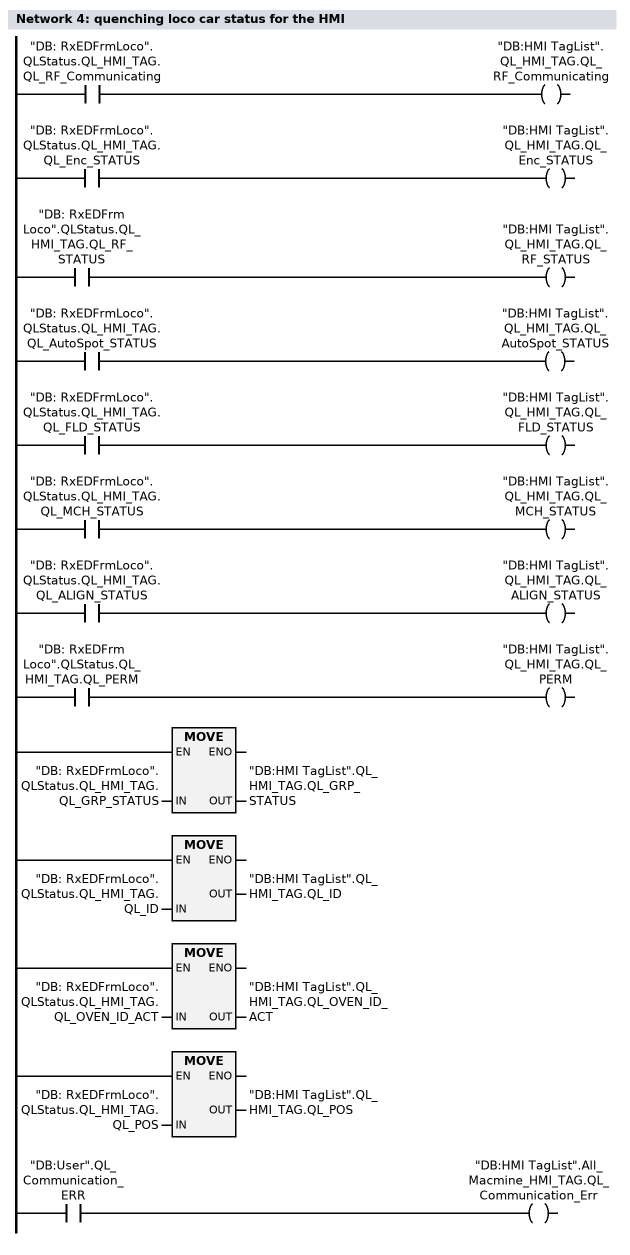
NETWORK
TITLE = quenching loco car status for the HMI
      A     "DB: RxEDFrmLoco".QLStatus.QL_HMI_TAG.QL_RF_Communicating;
      =     "DB:HMI TagList".QL_HMI_TAG.QL_RF_Communicating;
//..
      A     "DB: RxEDFrmLoco".QLStatus.QL_HMI_TAG.QL_Enc_STATUS;
      =     "DB:HMI TagList".QL_HMI_TAG.QL_Enc_STATUS;
//..
      A     "DB: RxEDFrmLoco".QLStatus.QL_HMI_TAG.QL_RF_STATUS;
      =     "DB:HMI TagList".QL_HMI_TAG.QL_RF_STATUS;
//..
      A     "DB: RxEDFrmLoco".QLStatus.QL_HMI_TAG.QL_AutoSpot_STATUS;
      =     "DB:HMI TagList".QL_HMI_TAG.QL_AutoSpot_STATUS;
//..
      A     "DB: RxEDFrmLoco".QLStatus.QL_HMI_TAG.QL_FLD_STATUS;
      =     "DB:HMI TagList".QL_HMI_TAG.QL_FLD_STATUS;
//..
      A     "DB: RxEDFrmLoco".QLStatus.QL_HMI_TAG.QL_MCH_STATUS;
      =     "DB:HMI TagList".QL_HMI_TAG.QL_MCH_STATUS;
//...
      A     "DB: RxEDFrmLoco".QLStatus.QL_HMI_TAG.QL_ALIGN_STATUS;
      =     "DB:HMI TagList".QL_HMI_TAG.QL_ALIGN_STATUS;
//..
      A     "DB: RxEDFrmLoco".QLStatus.QL_HMI_TAG.QL_PERM;
      =     "DB:HMI TagList".QL_HMI_TAG.QL_PERM;
//..
      L     "DB: RxEDFrmLoco".QLStatus.QL_HMI_TAG.QL_GRP_STATUS;
      T     "DB:HMI TagList".QL_HMI_TAG.QL_GRP_STATUS;
//..
      L     "DB: RxEDFrmLoco".QLStatus.QL_HMI_TAG.QL_ID;
      T     "DB:HMI TagList".QL_HMI_TAG.QL_ID;
//...
      L     "DB: RxEDFrmLoco".QLStatus.QL_HMI_TAG.QL_OVEN_ID_ACT;
      T     "DB:HMI TagList".QL_HMI_TAG.QL_OVEN_ID_ACT;
//..
      L     "DB: RxEDFrmLoco".QLStatus.QL_HMI_TAG.QL_POS;
      T     "DB:HMI TagList".QL_HMI_TAG.QL_POS;
//..
      A     "DB:User".QL_Communication_ERR;
      =     "DB:HMI TagList".All_Macmine_HMI_TAG.QL_Communication_Err;
///////////...............
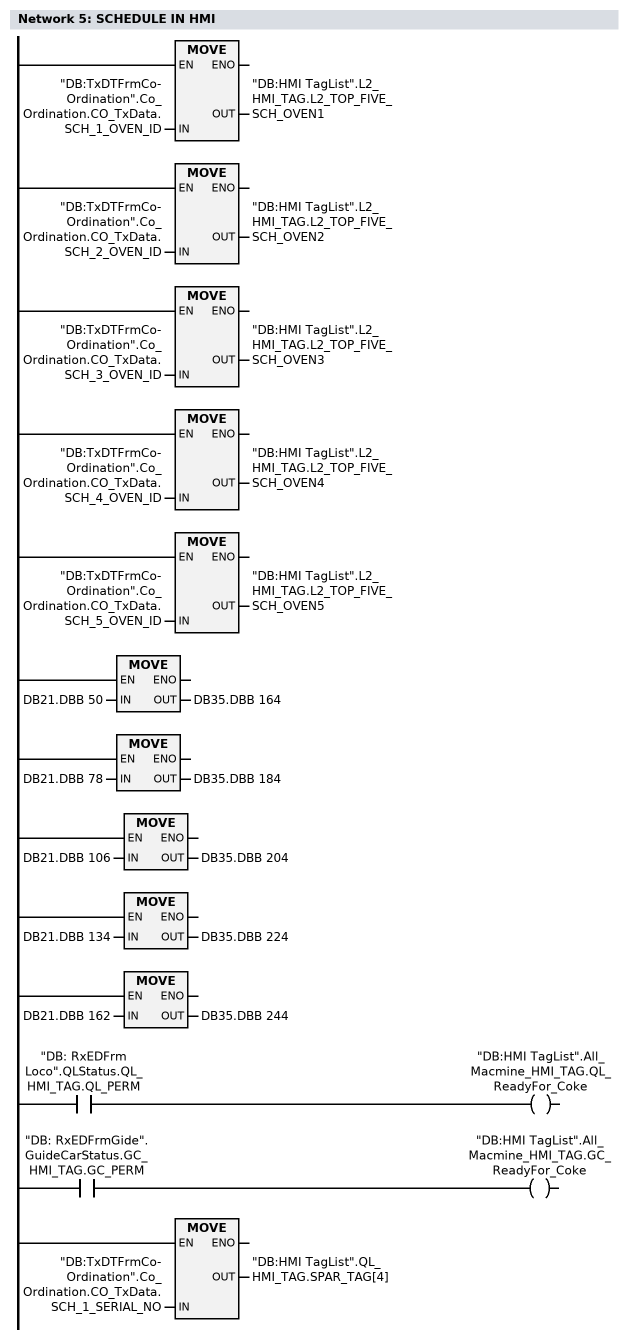
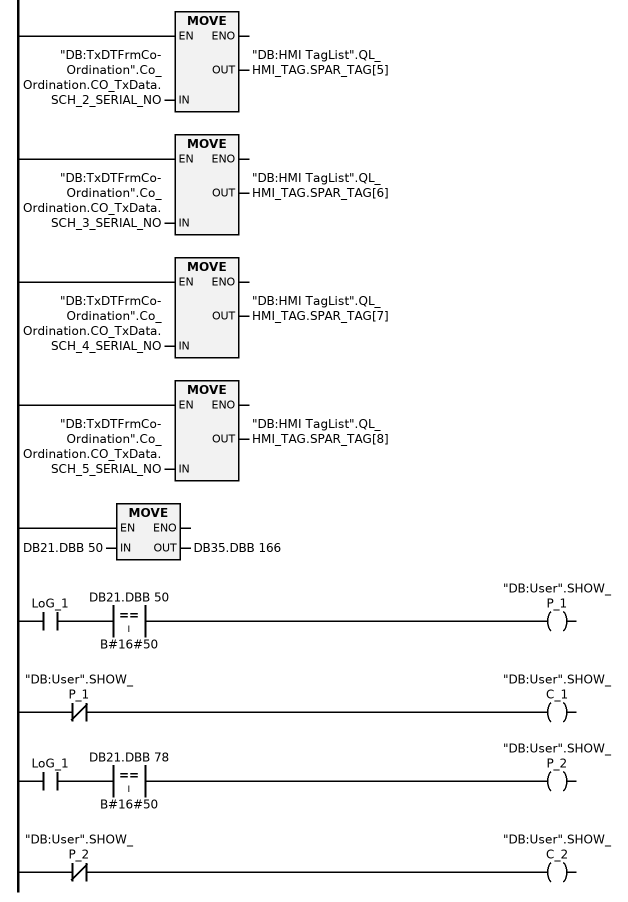
NETWORK
TITLE = SCHEDULE IN HMI
      L     "DB:TxDTFrmCo-Ordination".Co_Ordination.CO_TxData.SCH_1_OVEN_ID;
      T     "DB:HMI TagList".L2_HMI_TAG.L2_TOP_FIVE_SCH_OVEN1;
//..
      L     "DB:TxDTFrmCo-Ordination".Co_Ordination.CO_TxData.SCH_2_OVEN_ID;
      T     "DB:HMI TagList".L2_HMI_TAG.L2_TOP_FIVE_SCH_OVEN2;
//..
      L     "DB:TxDTFrmCo-Ordination".Co_Ordination.CO_TxData.SCH_3_OVEN_ID;
      T     "DB:HMI TagList".L2_HMI_TAG.L2_TOP_FIVE_SCH_OVEN3;
//..
      L     "DB:TxDTFrmCo-Ordination".Co_Ordination.CO_TxData.SCH_4_OVEN_ID;
      T     "DB:HMI TagList".L2_HMI_TAG.L2_TOP_FIVE_SCH_OVEN4;
//..
      L     "DB:TxDTFrmCo-Ordination".Co_Ordination.CO_TxData.SCH_5_OVEN_ID;
      T     "DB:HMI TagList".L2_HMI_TAG.L2_TOP_FIVE_SCH_OVEN5;
//..
      L     DB21.DBB 50;
      T     DB35.DBB 164;
//..
      L     DB21.DBB 78;
      T     DB35.DBB 184;
//..
      L     DB21.DBB 106;
      T     DB35.DBB 204;
//..
      L     DB21.DBB 134;
      T     DB35.DBB 224;
//..
      L     DB21.DBB 162;
      T     DB35.DBB 244;
//...
//...--------QL AND GC PERMISS MOVE TO HMI---------//......
      A     "DB: RxEDFrmLoco".QLStatus.QL_HMI_TAG.QL_PERM;
      =     "DB:HMI TagList".All_Macmine_HMI_TAG.QL_ReadyFor_Coke;
//..
      A     "DB: RxEDFrmGide".GuideCarStatus.GC_HMI_TAG.GC_PERM;
      =     "DB:HMI TagList".All_Macmine_HMI_TAG.GC_ReadyFor_Coke;
//..-------------START OVEEN NO INDICATION TO HMI-----------------------...//
      L     "DB:TxDTFrmCo-Ordination".Co_Ordination.CO_TxData.SCH_1_SERIAL_NO;
      T     "DB:HMI TagList".QL_HMI_TAG.SPAR_TAG[4];
//..
      L     "DB:TxDTFrmCo-Ordination".Co_Ordination.CO_TxData.SCH_2_SERIAL_NO;
      T     "DB:HMI TagList".QL_HMI_TAG.SPAR_TAG[5];
//..
      L     "DB:TxDTFrmCo-Ordination".Co_Ordination.CO_TxData.SCH_3_SERIAL_NO;
      T     "DB:HMI TagList".QL_HMI_TAG.SPAR_TAG[6];
//..
      L     "DB:TxDTFrmCo-Ordination".Co_Ordination.CO_TxData.SCH_4_SERIAL_NO;
      T     "DB:HMI TagList".QL_HMI_TAG.SPAR_TAG[7];
//..
      L     "DB:TxDTFrmCo-Ordination".Co_Ordination.CO_TxData.SCH_5_SERIAL_NO;
      T     "DB:HMI TagList".QL_HMI_TAG.SPAR_TAG[8];
//..
      L     DB21.DBB 50;
      T     DB35.DBB 166;
//..-------------END OVEEN NO INDICATION TO HMI-----------------------...//
//..    show P&C indication for oven no 1&2 in schedule
      A     "LoG_1";
      A(;
      L     DB21.DBB 50;
      L     B#16#50;
      ==I;
      );
      =     "DB:User".SHOW_P_1;
//.. show c indication if not p
      AN    "DB:User".SHOW_P_1;
      =     "DB:User".SHOW_C_1;
//..show P&C indication for oven no 2 in schedule
      A     "LoG_1";
      A(;
      L     DB21.DBB 78;
      L     B#16#50;
      ==I;
      );
      =     "DB:User".SHOW_P_2;
//..
      AN    "DB:User".SHOW_P_2;
      =     "DB:User".SHOW_C_2;
//...========================END===========================================
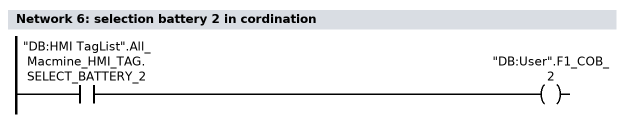
NETWORK
TITLE = selection battery 2 in cordination
      A     "DB:HMI TagList".All_Macmine_HMI_TAG.SELECT_BATTERY_2;
      =     "DB:User".F1_COB_2;
END_FUNCTION

FUNCTION "FC:FreqChanging" : VOID	// FC 28
VERSION : 0.1
VAR_INPUT
  F1_Set : BOOL ;	//Frequency Satting F1 Battery#1
  Offline : BOOL ;	//Machine Offline Mode
END_VAR
VAR_OUTPUT
  ModemFreQ_Set_Don : BOOL ;	//Modem Frequency Set OK
  ModemFreQ_Set_Err : BOOL ;	//Modem Frequency not Set
END_VAR
BEGIN
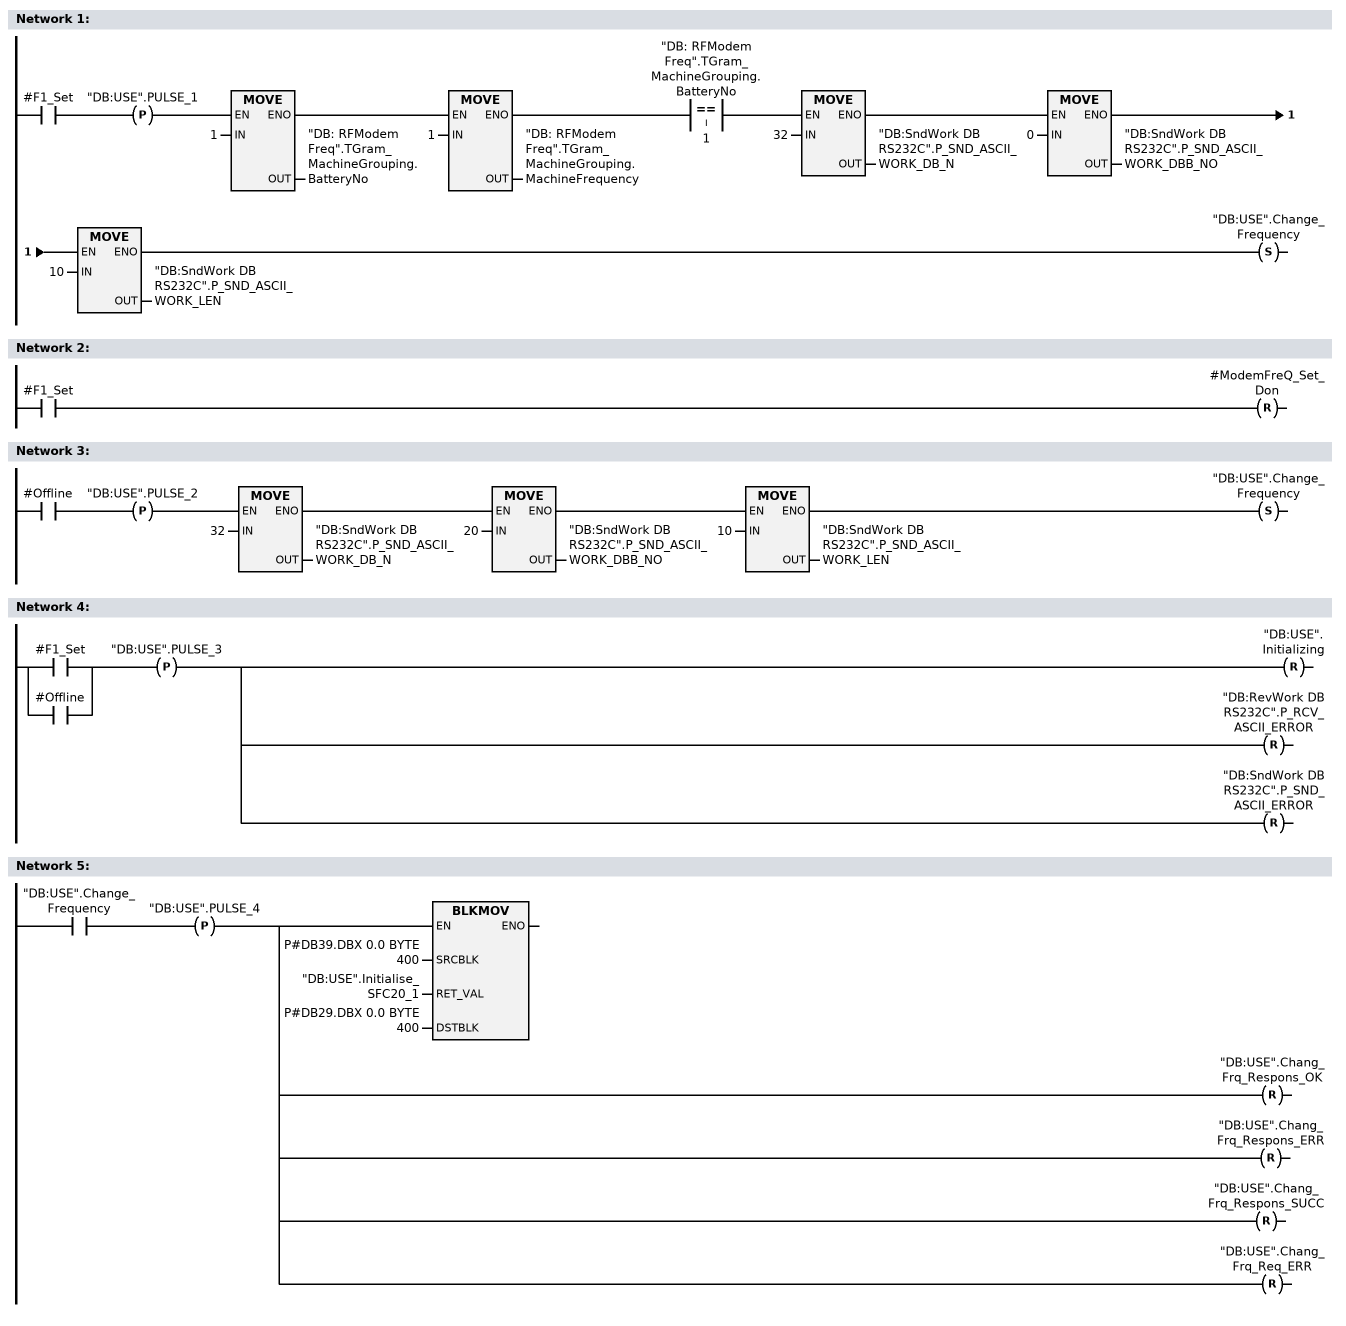
NETWORK
TITLE =
//Change Frequency Request: Initializing        
      A(;
      A(;
      A(;
      A(;
      A     #F1_Set;
      FP    "DB:USE".PULSE_1;
      JNB   _001;
      L     1;
      T     "DB: RFModem Freq".TGram_MachineGrouping.BatteryNo;
      SET;
      SAVE;
      CLR;
_001: A     BR;
      );
      JNB   _002;
      L     1;
      T     "DB: RFModem Freq".TGram_MachineGrouping.MachineFrequency;
      SET;
      SAVE;
      CLR;
_002: A     BR;
      );
      A(;
      L     "DB: RFModem Freq".TGram_MachineGrouping.BatteryNo;
      L     1;
      ==I;
      );
      JNB   _003;
      L     32;
      T     "DB:SndWork DB RS232C".P_SND_ASCII_WORK_DB_N;
      SET;
      SAVE;
      CLR;
_003: A     BR;
      );
      JNB   _004;
      L     0;
      T     "DB:SndWork DB RS232C".P_SND_ASCII_WORK_DBB_NO;
      SET;
      SAVE;
      CLR;
_004: A     BR;
      );
      JNB   _005;
      L     10;
      T     "DB:SndWork DB RS232C".P_SND_ASCII_WORK_LEN;
      SET;
      SAVE;
      CLR;
_005: A     BR;
      S     "DB:USE".Change_Frequency;
NETWORK
TITLE =
      A     #F1_Set;
      R     #ModemFreQ_Set_Don;
NETWORK
TITLE =
//Change Frequency Request: Initializing  
      A(;
      A(;
      A     #Offline;
      FP    "DB:USE".PULSE_2;
      JNB   _006;
      L     32;
      T     "DB:SndWork DB RS232C".P_SND_ASCII_WORK_DB_N;
      SET;
      SAVE;
      CLR;
_006: A     BR;
      );
      JNB   _007;
      L     20;
      T     "DB:SndWork DB RS232C".P_SND_ASCII_WORK_DBB_NO;
      SET;
      SAVE;
      CLR;
_007: A     BR;
      );
      JNB   _008;
      L     10;
      T     "DB:SndWork DB RS232C".P_SND_ASCII_WORK_LEN;
      SET;
      SAVE;
      CLR;
_008: A     BR;
      S     "DB:USE".Change_Frequency;
NETWORK
TITLE =
//Change Frequency Request: Initializing
      A(;
      O     #F1_Set;
      O     #Offline;
      );
      FP    "DB:USE".PULSE_3;
      R     "DB:USE".Initializing;
      R     "DB:RevWork DB RS232C".P_RCV_ASCII_ERROR;
      R     "DB:SndWork DB RS232C".P_SND_ASCII_ERROR;
NETWORK
TITLE =
//Change Frequency Request: Clearing Response Area & ACK/NACK
      A     "DB:USE".Change_Frequency;
      FP    "DB:USE".PULSE_4;
      =     L 0.0;
      A     L 0.0;
      JNB   _009;
      CALL  "BLKMOV" (
           SRCBLK                   := P#DB39.DBX 0.0 BYTE 400,
           RET_VAL                  := "DB:USE".Initialise_SFC20_1,
           DSTBLK                   := P#DB29.DBX 0.0 BYTE 400);
_009: NOP   0;
      A     L 0.0;
      BLD   102;
      R     "DB:USE".Chang_Frq_Respons_OK;
      A     L 0.0;
      BLD   102;
      R     "DB:USE".Chang_Frq_Respons_ERR;
      A     L 0.0;
      BLD   102;
      R     "DB:USE".Chang_Frq_Respons_SUCC;
      A     L 0.0;
      BLD   102;
      R     "DB:USE".Chang_Frq_Req_ERR;
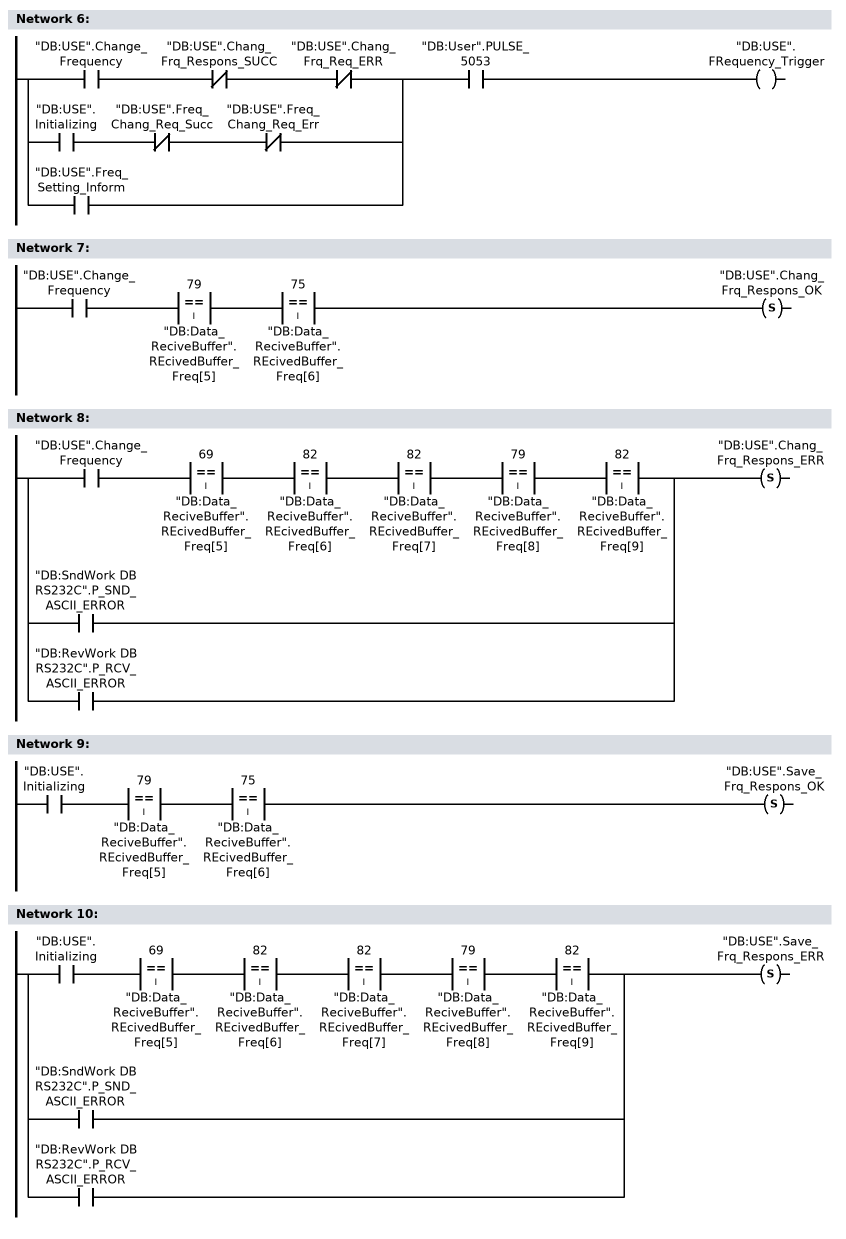
NETWORK
TITLE =
//Change Frequency Request: Try Sending To CP
      A(;
      A     "DB:USE".Change_Frequency;
      AN    "DB:USE".Chang_Frq_Respons_SUCC;
      AN    "DB:USE".Chang_Frq_Req_ERR;
      O;
      A     "DB:USE".Initializing;
      AN    "DB:USE".Freq_Chang_Req_Succ;
      AN    "DB:USE".Freq_Chang_Req_Err;
      O     "DB:USE".Freq_Setting_Inform;
      );
      A     "DB:User".PULSE_5053;
      =     "DB:USE".FRequency_Trigger;
NETWORK
TITLE =
//Change Frequency Request: ACK Response Evaluation (OK Recieved In Empty DB, 
//Succesfull Sent Condition Is Implied Otherwise We Will Not Get Response)
      A     "DB:USE".Change_Frequency;
      A(;
      L     79;	// ASCII 79 = 'O'
      L     "DB:Data_ReciveBuffer".REcivedBuffer_Freq[5];
      ==I;
      );
      A(;
      L     75;	// ASCII 75 = 'K'
      L     "DB:Data_ReciveBuffer".REcivedBuffer_Freq[6];
      ==I;
      );
      S     "DB:USE".Chang_Frq_Respons_OK;
NETWORK
TITLE =
//Change Frequency Request: NACK Response Evaluation (Error Recieved In Empty DB 
//Or Error During Tx Or Rx)
      A     "DB:USE".Change_Frequency;
      A(;
      L     69;	// ASCII 69 = 'E'
      L     "DB:Data_ReciveBuffer".REcivedBuffer_Freq[5];
      ==I;
      );
      A(;
      L     82;	// ASCII 82 = 'R'
      L     "DB:Data_ReciveBuffer".REcivedBuffer_Freq[6];
      ==I;
      );
      A(;
      L     82;	// ASCII 82 = 'R'
      L     "DB:Data_ReciveBuffer".REcivedBuffer_Freq[7];
      ==I;
      );
      A(;
      L     79;	// ASCII 79 = 'O'
      L     "DB:Data_ReciveBuffer".REcivedBuffer_Freq[8];
      ==I;
      );
      A(;
      L     82;	// ASCII 82 = 'R'
      L     "DB:Data_ReciveBuffer".REcivedBuffer_Freq[9];
      ==I;
      );
      O     "DB:SndWork DB RS232C".P_SND_ASCII_ERROR;
      O     "DB:RevWork DB RS232C".P_RCV_ASCII_ERROR;
      S     "DB:USE".Chang_Frq_Respons_ERR;
NETWORK
TITLE =
//Save Frequency Request: ACK Response Evaluation (OK Recieved In Empty DB, 
//Succesfull Sent Condition Is Implied Otherwise We Will Not Get Response)
      A     "DB:USE".Initializing;
      A(;
      L     79;	// ASCII 79 = 'O'
      L     "DB:Data_ReciveBuffer".REcivedBuffer_Freq[5];
      ==I;
      );
      A(;
      L     75;	// ASCII 75 = 'K'
      L     "DB:Data_ReciveBuffer".REcivedBuffer_Freq[6];
      ==I;
      );
      S     "DB:USE".Save_Frq_Respons_OK;
NETWORK
TITLE =
//Save Frequency Request: NACK Response Evaluation (Error Recieved In Empty DB 
//Or Error During Tx Or Rx)
      A     "DB:USE".Initializing;
      A(;
      L     69;	// ASCII 69 = 'E'
      L     "DB:Data_ReciveBuffer".REcivedBuffer_Freq[5];
      ==I;
      );
      A(;
      L     82;	// ASCII 82 = 'R'
      L     "DB:Data_ReciveBuffer".REcivedBuffer_Freq[6];
      ==I;
      );
      A(;
      L     82;	// ASCII 82 = 'R'
      L     "DB:Data_ReciveBuffer".REcivedBuffer_Freq[7];
      ==I;
      );
      A(;
      L     79;	// ASCII 79 = 'O'
      L     "DB:Data_ReciveBuffer".REcivedBuffer_Freq[8];
      ==I;
      );
      A(;
      L     82;	// ASCII 82 = 'R'
      L     "DB:Data_ReciveBuffer".REcivedBuffer_Freq[9];
      ==I;
      );
      O     "DB:SndWork DB RS232C".P_SND_ASCII_ERROR;
      O     "DB:RevWork DB RS232C".P_RCV_ASCII_ERROR;
      S     "DB:USE".Save_Frq_Respons_ERR;
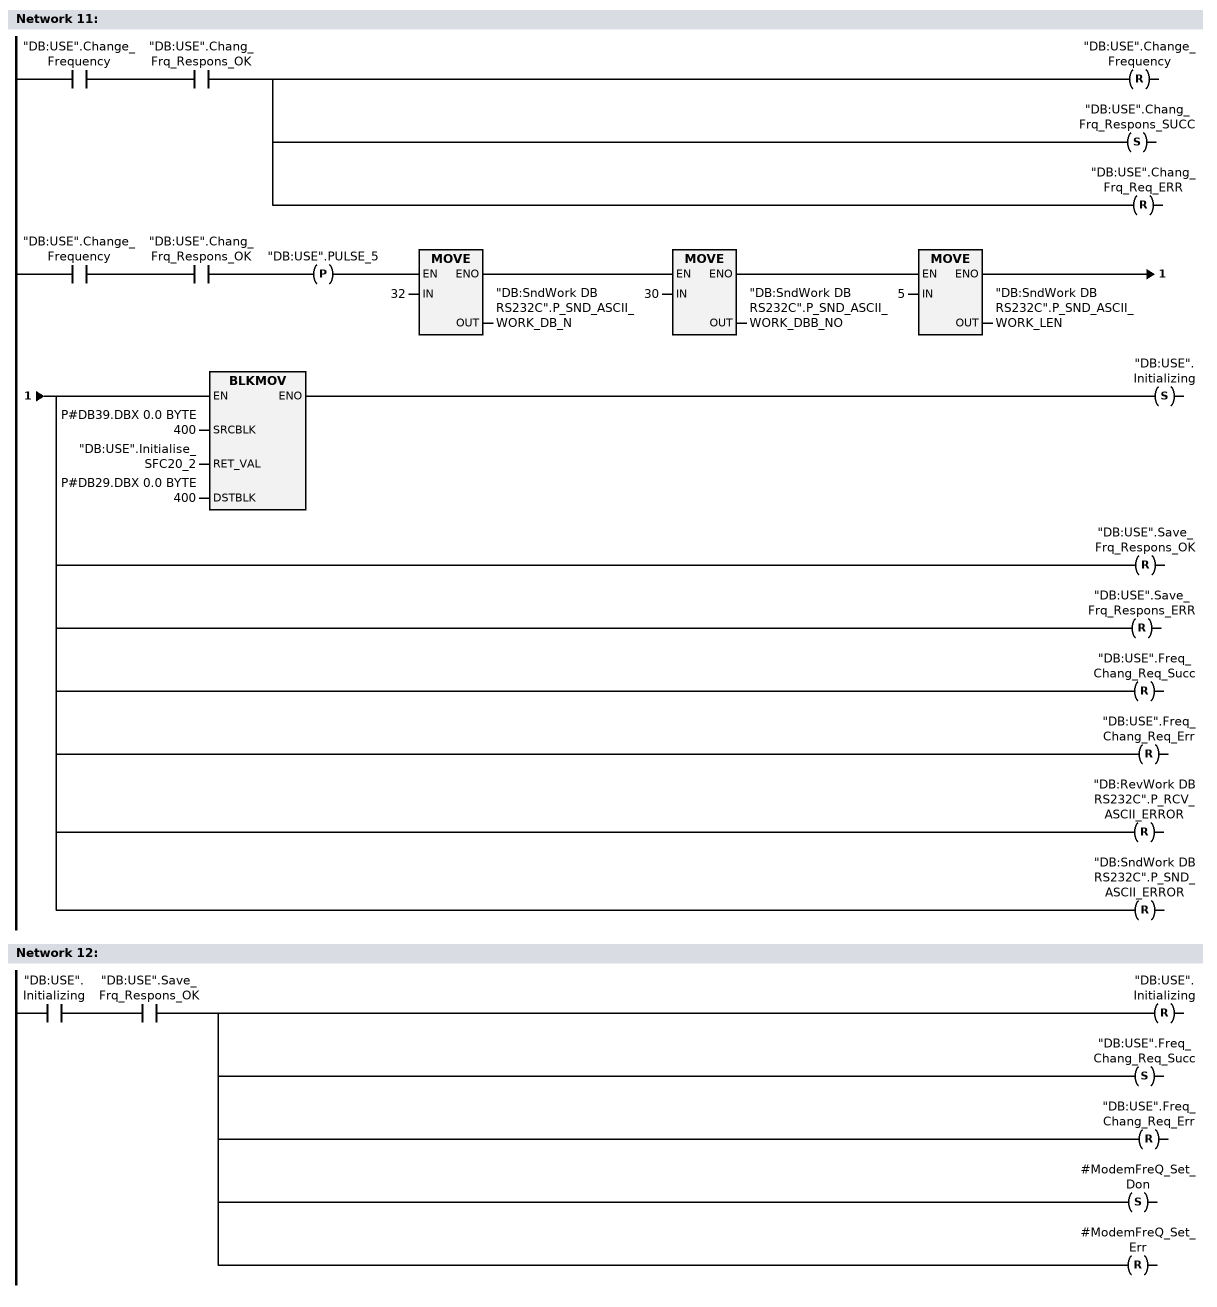
NETWORK
TITLE =
//Change Frequency Request: Success (Sent & ACK Recieved)
      A     "DB:USE".Change_Frequency;
      A     "DB:USE".Chang_Frq_Respons_OK;
      =     L 0.0;
      A     L 0.0;
      BLD   102;
      R     "DB:USE".Change_Frequency;
      A     L 0.0;
      BLD   102;
      S     "DB:USE".Chang_Frq_Respons_SUCC;
      A     L 0.0;
      BLD   102;
      R     "DB:USE".Chang_Frq_Req_ERR;
      A(;
      A(;
      A     L 0.0;
      FP    "DB:USE".PULSE_5;
      JNB   _00a;
      L     32;
      T     "DB:SndWork DB RS232C".P_SND_ASCII_WORK_DB_N;
      SET;
      SAVE;
      CLR;
_00a: A     BR;
      );
      JNB   _00b;
      L     30;
      T     "DB:SndWork DB RS232C".P_SND_ASCII_WORK_DBB_NO;
      SET;
      SAVE;
      CLR;
_00b: A     BR;
      );
      JNB   _00c;
      L     5;
      T     "DB:SndWork DB RS232C".P_SND_ASCII_WORK_LEN;
      SET;
      SAVE;
      CLR;
_00c: A     BR;
      =     L 0.1;
      A     L 0.1;
      JNB   _00d;
      CALL  "BLKMOV" (
           SRCBLK                   := P#DB39.DBX 0.0 BYTE 400,
           RET_VAL                  := "DB:USE".Initialise_SFC20_2,
           DSTBLK                   := P#DB29.DBX 0.0 BYTE 400);
_00d: A     BR;
      S     "DB:USE".Initializing;
      A     L 0.1;
      BLD   102;
      R     "DB:USE".Save_Frq_Respons_OK;
      A     L 0.1;
      BLD   102;
      R     "DB:USE".Save_Frq_Respons_ERR;
      A     L 0.1;
      BLD   102;
      R     "DB:USE".Freq_Chang_Req_Succ;
      A     L 0.1;
      BLD   102;
      R     "DB:USE".Freq_Chang_Req_Err;
      A     L 0.1;
      BLD   102;
      R     "DB:RevWork DB RS232C".P_RCV_ASCII_ERROR;
      A     L 0.1;
      BLD   102;
      R     "DB:SndWork DB RS232C".P_SND_ASCII_ERROR;
NETWORK
TITLE =
//Change Frequency Request: Success (Sent & ACK Recieved)
      A     "DB:USE".Initializing;
      A     "DB:USE".Save_Frq_Respons_OK;
      R     "DB:USE".Initializing;
      S     "DB:USE".Freq_Chang_Req_Succ;
      R     "DB:USE".Freq_Chang_Req_Err;
      S     #ModemFreQ_Set_Don;
      R     #ModemFreQ_Set_Err;
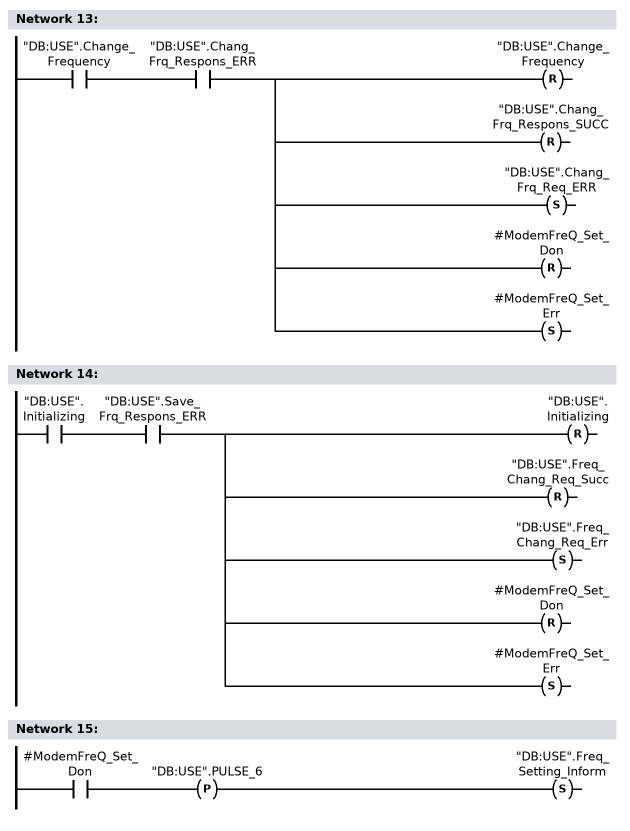
NETWORK
TITLE =
//Change Frequency Request: Error, Or NACK Recieved -> Set Error, Reset Done
      A     "DB:USE".Change_Frequency;
      A     "DB:USE".Chang_Frq_Respons_ERR;
      R     "DB:USE".Change_Frequency;
      R     "DB:USE".Chang_Frq_Respons_SUCC;
      S     "DB:USE".Chang_Frq_Req_ERR;
      R     #ModemFreQ_Set_Don;
      S     #ModemFreQ_Set_Err;
NETWORK
TITLE =
//Save Frequency Request: Error, Or NACK Recieved -> Set Error, Reset Done
      A     "DB:USE".Initializing;
      A     "DB:USE".Save_Frq_Respons_ERR;
      R     "DB:USE".Initializing;
      R     "DB:USE".Freq_Chang_Req_Succ;
      S     "DB:USE".Freq_Chang_Req_Err;
      R     #ModemFreQ_Set_Don;
      S     #ModemFreQ_Set_Err;
NETWORK
TITLE =
//Modem Frequency Set In F1= 436.2 Hz ;
//This Information Sand to Co-Ordination PLC Via RF
      A     #ModemFreQ_Set_Don;
      FP    "DB:USE".PULSE_6;
      S     "DB:USE".Freq_Setting_Inform;
NETWORK
TITLE =
NETWORK
TITLE =
NETWORK
TITLE =
      BE;
END_FUNCTION

FUNCTION "FC:RS232C RCV BLOCK" : VOID	// FC 29
VERSION : 0.1
VAR_INPUT
  CP_BassAdd : INT ;	//LADDR
  DB_No : INT ;	//DB No
  DBB_NO : INT ;	//Data Byte No
END_VAR
BEGIN
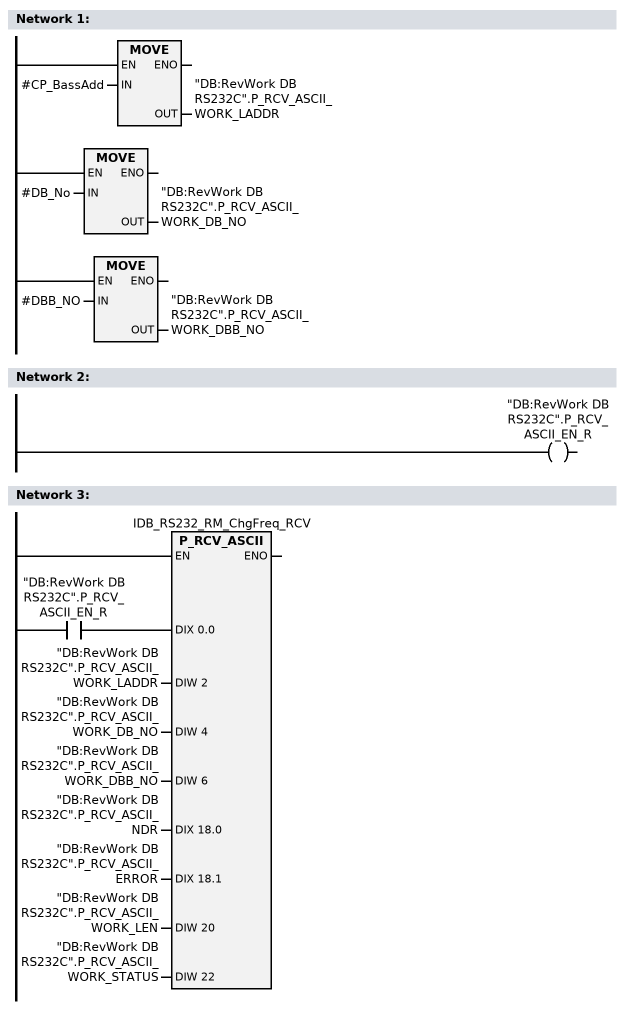
NETWORK
TITLE =
// ----------------------------
// Supply LADDR, DB_NO, DBB_NO
// ----------------------------
      L     #CP_BassAdd;
      T     "DB:RevWork DB RS232C".P_RCV_ASCII_WORK_LADDR;
//..
      L     #DB_No;
      T     "DB:RevWork DB RS232C".P_RCV_ASCII_WORK_DB_NO;
//..
      L     #DBB_NO;
      T     "DB:RevWork DB RS232C".P_RCV_ASCII_WORK_DBB_NO;
NETWORK
TITLE =
//// ------------------------
//// Enable Receive Data
//// ------------------------
//
      SET;
      =     "DB:RevWork DB RS232C".P_RCV_ASCII_EN_R;
NETWORK
TITLE =
//// ------------------------
//// P_RCV_RK with Instance-DB
//// ------------------------
//
      A     "DB:RevWork DB RS232C".P_RCV_ASCII_EN_R;
      =     L 0.0;
      BLD   103;
      CALL  "P_RCV_ASCII" , "IDB_RS232_RM_ChgFreq_RCV" (
           DIX 0.0                  := L 0.0,
           DIW 2                    := "DB:RevWork DB RS232C".P_RCV_ASCII_WORK_LADDR,
           DIW 4                    := "DB:RevWork DB RS232C".P_RCV_ASCII_WORK_DB_NO,
           DIW 6                    := "DB:RevWork DB RS232C".P_RCV_ASCII_WORK_DBB_NO,
           DIX 18.0                 := "DB:RevWork DB RS232C".P_RCV_ASCII_NDR,
           DIX 18.1                 := "DB:RevWork DB RS232C".P_RCV_ASCII_ERROR,
           DIW 20                   := "DB:RevWork DB RS232C".P_RCV_ASCII_WORK_LEN,
           DIW 22                   := "DB:RevWork DB RS232C".P_RCV_ASCII_WORK_STATUS);
      NOP   0;
NETWORK
TITLE =
// -------------------------------
// Check P_RCV_RK_NDR (Receive without error)
// -------------------------------
      AN    "DB:RevWork DB RS232C".P_RCV_ASCII_NDR;	//check P_RCV_RK_NDR
      JC    CHER;	//if P_RCV_RK_NDR equals FALSE, jump to CHER
//and check P_RCV_RK_ERROR
// -------------------------------
//  P_RCV_RK_NDR = 1 (Receive without error)
// -------------------------------
      L     "DB:RevWork DB RS232C".P_RCV_ASCII_WORK_CNT_OK;	//"Receive without error"
      +     1;	//increment counter
      T     "DB:RevWork DB RS232C".P_RCV_ASCII_WORK_CNT_OK;
      L     "DB:RevWork DB RS232C".P_RCV_ASCII_WORK_LEN;	//save RECEIVE-Length
      T     "DB:RevWork DB RS232C".P_RCV_ASCII_WORK_SAVE_LE;
      BE;
// -------------------------------
// Check "Receive with error"
// -------------------------------
CHER: AN    "DB:RevWork DB RS232C".P_RCV_ASCII_ERROR;	//check P_RCV_RK_ERROR
      BEC;	//if no error occured, jump to end
// -------------------------------
// "Receive with error"
// -------------------------------
      L     "DB:RevWork DB RS232C".P_RCV_ASCII_WORK_CNT_ERR;	//Error
      +     1;	//increment counter
      T     "DB:RevWork DB RS232C".P_RCV_ASCII_WORK_CNT_ERR;
// ----------------------------
// Save "P_RCV_RK_STATUS"
// ---------------------------- 
      L     "DB:RevWork DB RS232C".P_RCV_ASCII_WORK_STATUS;
      T     "DB:RevWork DB RS232C".P_RCV_WORK_STATUS_SAV;	//save P_RCV_RK_STATUS
      BE;
END_FUNCTION

FUNCTION "FC:RS232C SND BLOCK" : VOID	// FC 30
TITLE = Execute P_SND_ASCII-Jobs
VERSION : 0.1
VAR_INPUT
  SetFREQ : BOOL ;	//Req
  CP_BassAdd : INT ;	//LADDR
  DB_No : INT ;	//DB No
  DBB_NO : INT ;	//Data Byte No
  LEN : INT ;	//Lenth of Data
END_VAR
BEGIN
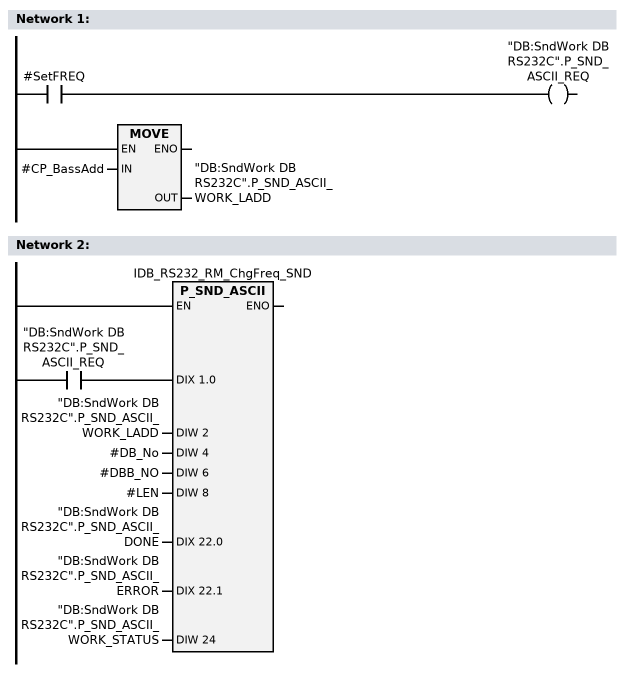
NETWORK
TITLE =
//------------------------
// Supply LADDR, DB_NO, DBB_NO, LEN
// ------------------------
// ------------------------
// Generate edge SEND_REQ
// ------------------------
      A     #SetFREQ;
      =     "DB:SndWork DB RS232C".P_SND_ASCII_REQ;	//Set SEND_REQ
//..
      L     #CP_BassAdd;	//LADDR
      T     "DB:SndWork DB RS232C".P_SND_ASCII_WORK_LADD;
NETWORK
TITLE =
//// ------------------------
//// SEND with Instance-DB
//// ------------------------
//
      A     "DB:SndWork DB RS232C".P_SND_ASCII_REQ;
      =     L 0.0;
      BLD   103;
      CALL  "P_SND_ASCII" , "IDB_RS232_RM_ChgFreq_SND" (
           DIX 1.0                  := L 0.0,
           DIW 2                    := "DB:SndWork DB RS232C".P_SND_ASCII_WORK_LADD,
           DIW 4                    := #DB_No,
           DIW 6                    := #DBB_NO,
           DIW 8                    := #LEN,
           DIX 22.0                 := "DB:SndWork DB RS232C".P_SND_ASCII_DONE,
           DIX 22.1                 := "DB:SndWork DB RS232C".P_SND_ASCII_ERROR,
           DIW 24                   := "DB:SndWork DB RS232C".P_SND_ASCII_WORK_STATUS);
      NOP   0;
NETWORK
TITLE =
// -------------------------------
// Check "Complete without error"
// -------------------------------
      AN    "DB:SndWork DB RS232C".P_SND_ASCII_DONE;	//check P_SND_RK_DONE
      JC    CHER;	//if P_SND_RK_DONE equals 0, jump to CHER
//and check P_SND_RK_ERROR
// -------------------------------
// "Complete without error"
//  P_SND_RK_DONE = 1
// -------------------------------
      L     "DB:SndWork DB RS232C".P_SND_ASCII_COUNTER_OK;	//"Complete without Error"
      +     1;	//increment counter
      T     "DB:SndWork DB RS232C".P_SND_ASCII_COUNTER_OK;
      NOP   0;
      NOP   0;	//further user functions
      NOP   0;
      BE;
// -------------------------------
// Check "Complete with error"
// P_SND_RK_ERROR = 1
// -------------------------------
CHER: AN    "DB:SndWork DB RS232C".P_SND_ASCII_ERROR;	//check P_SND_RK_ERROR
      BEC;	//if no error occured, jump to end
// -------------------------------
// "Complete with error"
// -------------------------------
      L     "DB:SndWork DB RS232C".P_SND_ASCII_COUNTER_ERR;	//"Complete with error"
      +     1;	//increment counter
      T     "DB:SndWork DB RS232C".P_SND_ASCII_COUNTER_ERR;
      L     "DB:SndWork DB RS232C".P_SND_ASCII_WORK_STATUS;
      T     "DB:SndWork DB RS232C".P_SND_WORK_STATUS_SAV;	//save STATUS
      NOP   0;
      NOP   0;	//Error-Handling
      NOP   0;
      BE;
NETWORK
TITLE =
END_FUNCTION

FUNCTION "FC: RdAutoSPOT" : VOID	// FC 31
//This function reads AutoSPOT Telegrams & performs following jobs
//
//1. Detect Packets Recieved, Verify Packets Recieved & Detect No Data 
//(LinkFail). Link fail is a condition when no data or invalid data (except unit 
//id & crc matching) occurs for 8 seconds. Link fail is availaible as function 
//output.
//2. Extract plate address from recieved information packet when aligned and not 
//linkfail and add 100 constant to update oven id output. In case of LinkFail 
//last oven id is retained as output (Note: Same locations like ovens, 
//quenching-towers etc for both batteries shall have different plate number 
//unlike in VSP)
//3. Extract unit id from any packet when not linkfail and update unit id output. 
//In case of LinkFail last unit id is retained as output 
//4. Extract aligned, left aligned and right aligned from any packet recieved and 
//not linkfail
//5. If Detects Machine In Wrong Battery from Currently Selected Battery using 
//Marker Plate Value
//
//Reserved:
//- DB31: AutoSPOT Communication -> Data, Status and Results Are Stored Here
//- DB71: Instance DB for AutoSPOT Communication
//- C127: Timeout Detection Counter
AUTHOR : SKD
NAME : CDSPL
VERSION : 0.1
VAR_INPUT
  Enable : BOOL ;	//Enable AutoSPOT Reading
  CPAddr : INT ;	//Base Address of RS485 Card (CP341)
  SelBatt : INT ;	//Currently Selected Battery {0 - Offline, 1-Battery #1, 2-Battery #2}
END_VAR
VAR_OUTPUT
  OvenID : INT ;	//Oven Number Machine Is Aligned At.
  UnitID : INT ;	//UnitID Of Connected AutoSPOT H/w
  Aligned : BOOL ;	//True = If Both S9/Left & S10/Right Markers Are Blocked
  S9Aligned : BOOL ;	//True = If S9/Left Marker Is Blocked
  S10Aligned : BOOL ;	//True = If S10/Right Marker Is Blocked
  LinkFail : BOOL ;	//True = If Communication Error, Bad Data Etc.
  McInWrongBatt : BOOL ;	//True If Machine Movement In Wrong Battery
END_VAR
VAR_TEMP
  tCtrCV : WORD ;
  tOvenID : INT ;
END_VAR
BEGIN
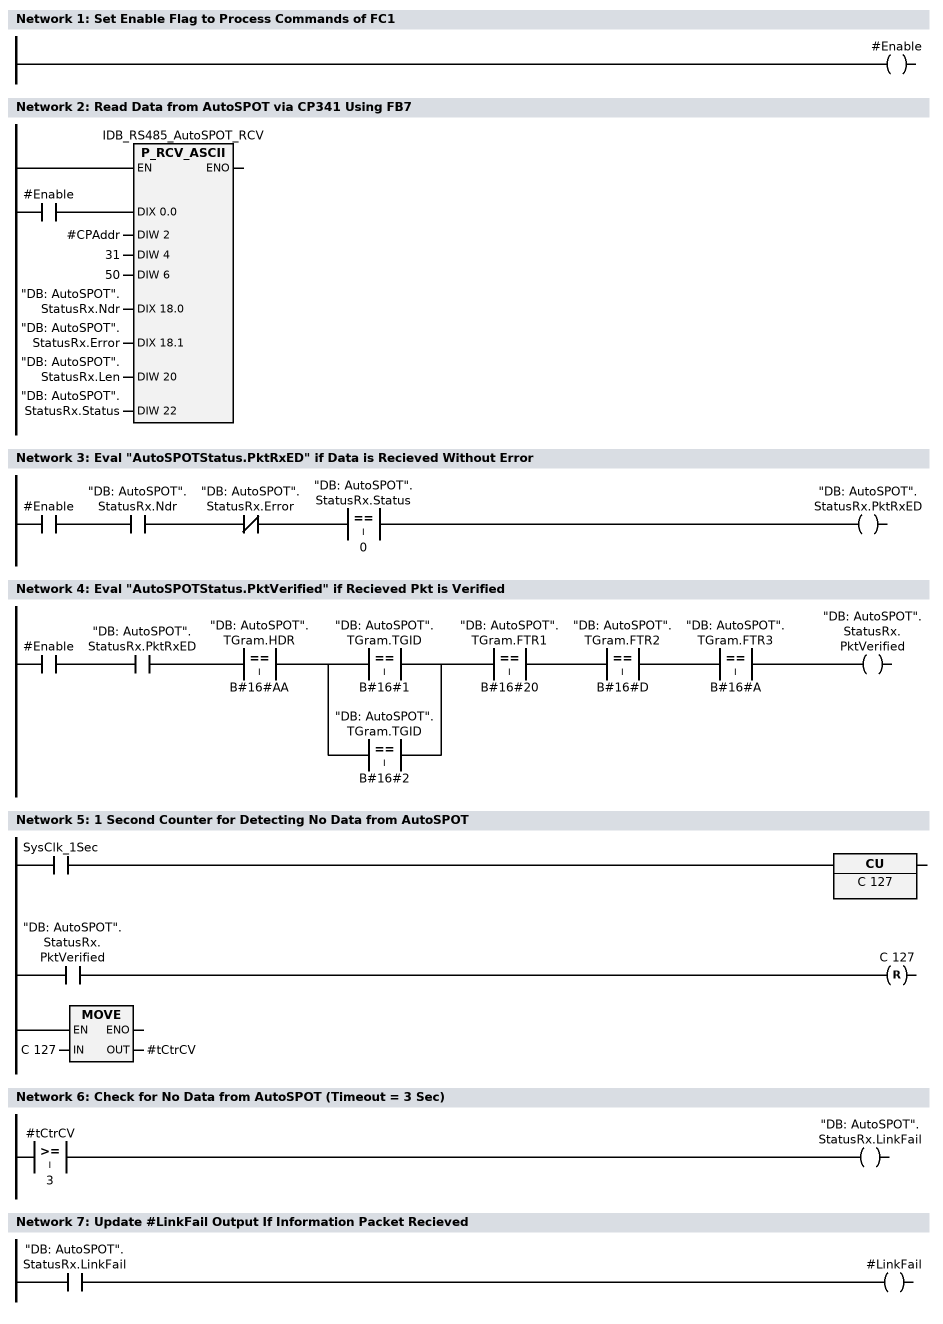
NETWORK
TITLE = Set Enable Flag to Process Commands of FC1
//Set Enable Flag to Process Commands of FC1
      SET;
      =     #Enable;
NETWORK
TITLE = Read Data from AutoSPOT via CP341 Using FB7
//Read Data from AutoSPOT via CP341 Using FB7
      A     #Enable;
      =     L 4.0;
      BLD   103;
      CALL  "P_RCV_ASCII" , "IDB_RS485_AutoSPOT_RCV" (
           DIX 0.0                  := L 4.0,
           DIW 2                    := #CPAddr,
           DIW 4                    := 31,
           DIW 6                    := 50,
           DIX 18.0                 := "DB: AutoSPOT".StatusRx.Ndr,
           DIX 18.1                 := "DB: AutoSPOT".StatusRx.Error,
           DIW 20                   := "DB: AutoSPOT".StatusRx.Len,
           DIW 22                   := "DB: AutoSPOT".StatusRx.Status);
      NOP   0;
NETWORK
TITLE = Eval "AutoSPOTStatus.PktRxED" if Data is Recieved Without Error
//Eval "AutoSPOTStatus.PktRxED" if Data is Recieved Without Error
//(Condition: Ndr And !Error AND Status=0) 
      A     #Enable;
      A     "DB: AutoSPOT".StatusRx.Ndr;
      AN    "DB: AutoSPOT".StatusRx.Error;
      A(;
      L     "DB: AutoSPOT".StatusRx.Status;
      L     0;
      ==I;
      );
      =     "DB: AutoSPOT".StatusRx.PktRxED;
NETWORK
TITLE = Eval "AutoSPOTStatus.PktVerified" if Recieved Pkt is Verified
//Eval "AutoSPOTStatus.PktVerified" if Recieved Pkt is Verified
//(Condition: Match HDR, TGID, & FTR1 to FTR3; Ignore CRC)
      A     #Enable;
      A     "DB: AutoSPOT".StatusRx.PktRxED;
//Match HDR
      A(;
      L     "DB: AutoSPOT".TGram.HDR;
      L     B#16#AA;
      ==I;
      );
//Match TGID
      A(;
      O(;
      L     "DB: AutoSPOT".TGram.TGID;
      L     B#16#1;
      ==I;
      );
      O(;
      L     "DB: AutoSPOT".TGram.TGID;
      L     B#16#2;
      ==I;
      );
      );
//Match FTR1
      A(;
      L     "DB: AutoSPOT".TGram.FTR1;
      L     B#16#20;
      ==I;
      );
//Match FTR2
      A(;
      L     "DB: AutoSPOT".TGram.FTR2;
      L     B#16#D;
      ==I;
      );
//Match FTR3
      A(;
      L     "DB: AutoSPOT".TGram.FTR3;
      L     B#16#A;
      ==I;
      );
      =     "DB: AutoSPOT".StatusRx.PktVerified;
NETWORK
TITLE = 1 Second Counter for Detecting No Data from AutoSPOT
//1 Second Counter for Detecting No Data from AutoSPOT
      A     "SysClk_1Sec";
      CU    C 127;
      BLD   101;
      NOP   0;
      NOP   0;
      A     "DB: AutoSPOT".StatusRx.PktVerified;
      R     C 127;
      L     C 127;
      T     #tCtrCV;
      NOP   0;
      NOP   0;
NETWORK
TITLE = Check for No Data from AutoSPOT (Timeout = 3 Sec)
//Check for No Data from AutoSPOT (Timeout = 3 Sec)
//Match Counter > 3 Seconds
      L     #tCtrCV;
      L     3;
      >=I;
      =     "DB: AutoSPOT".StatusRx.LinkFail;
NETWORK
TITLE = Update #LinkFail Output If Information Packet Recieved
//Update #LinkFail Output If Information Packet Recieved
      A     "DB: AutoSPOT".StatusRx.LinkFail;
      =     #LinkFail;
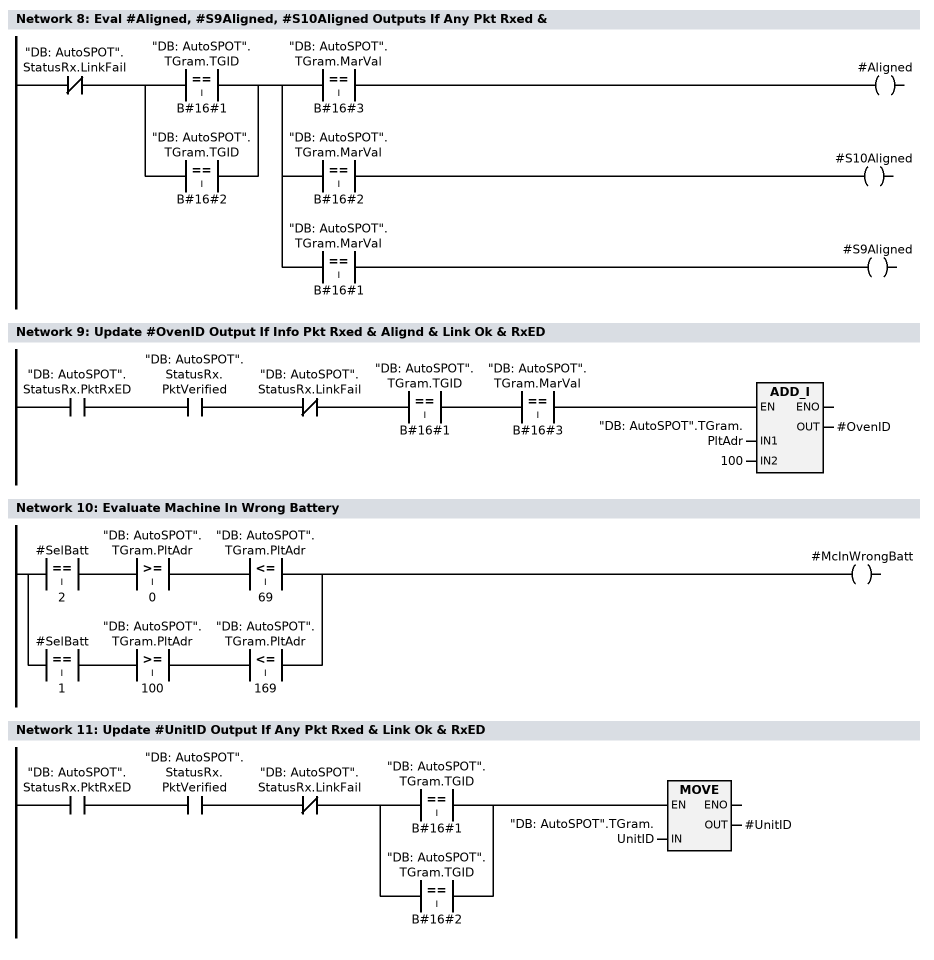
NETWORK
TITLE = Eval #Aligned, #S9Aligned, #S10Aligned Outputs If Any Pkt Rxed &
//Eval #Aligned, #S9Aligned, #S10Aligned Outputs If Any Pkt Rxed & Link Is Ok
      AN    "DB: AutoSPOT".StatusRx.LinkFail;
      A(;
      O(;
      L     "DB: AutoSPOT".TGram.TGID;
      L     B#16#1;
      ==I;
      );
      O(;
      L     "DB: AutoSPOT".TGram.TGID;
      L     B#16#2;
      ==I;
      );
      );
      =     L 2.0;
      A     L 2.0;
      A(;
      L     "DB: AutoSPOT".TGram.MarVal;
      L     B#16#3;
      ==I;
      );
      =     #Aligned;
      A     L 2.0;
      A(;
      L     "DB: AutoSPOT".TGram.MarVal;
      L     B#16#2;
      ==I;
      );
      =     #S10Aligned;
      A     L 2.0;
      A(;
      L     "DB: AutoSPOT".TGram.MarVal;
      L     B#16#1;
      ==I;
      );
      =     #S9Aligned;
NETWORK
TITLE = Update #OvenID Output If Info Pkt Rxed & Alignd & Link Ok & RxED
//Update #OvenID Output If Info Pkt Rxed & Alignd & Link Ok & RxED
      A     "DB: AutoSPOT".StatusRx.PktRxED;
      A     "DB: AutoSPOT".StatusRx.PktVerified;
      AN    "DB: AutoSPOT".StatusRx.LinkFail;
      A(;
      L     "DB: AutoSPOT".TGram.TGID;
      L     B#16#1;
      ==I;
      );
      A(;
      L     "DB: AutoSPOT".TGram.MarVal;
      L     B#16#3;
      ==I;
      );
      JNB   _002;
      L     "DB: AutoSPOT".TGram.PltAdr;
      L     100;
      +I;
      T     #OvenID;
_002: NOP   0;
NETWORK
TITLE = Evaluate Machine In Wrong Battery
//If Selection = Battery #2/1 && PlateValue from #0/100-69/169 => Machine Is 
//Moved In Wrong Battery
      A(;
      L     #SelBatt;
      L     2;
      ==I;
      );
      A(;
      L     "DB: AutoSPOT".TGram.PltAdr;
      L     0;
      >=I;
      );
      A(;
      L     "DB: AutoSPOT".TGram.PltAdr;
      L     69;
      <=I;
      );
      O;
      A(;
      L     #SelBatt;
      L     1;
      ==I;
      );
      A(;
      L     "DB: AutoSPOT".TGram.PltAdr;
      L     100;
      >=I;
      );
      A(;
      L     "DB: AutoSPOT".TGram.PltAdr;
      L     169;
      <=I;
      );
      =     #McInWrongBatt;
NETWORK
TITLE = Update #UnitID Output If Any Pkt Rxed & Link Ok & RxED
//Update #UnitID Output If Any Pkt Rxed & Link Ok & RxED
      A     "DB: AutoSPOT".StatusRx.PktRxED;
      A     "DB: AutoSPOT".StatusRx.PktVerified;
      AN    "DB: AutoSPOT".StatusRx.LinkFail;
      A(;
      O(;
      L     "DB: AutoSPOT".TGram.TGID;
      L     B#16#1;
      ==I;
      );
      O(;
      L     "DB: AutoSPOT".TGram.TGID;
      L     B#16#2;
      ==I;
      );
      );
      JNB   _001;
      L     "DB: AutoSPOT".TGram.UnitID;
      T     #UnitID;
_001: NOP   0;
NETWORK
TITLE = Error Status Handling
//Error Status Handling
// -------------------------------
// Check "Receive without error"
// -------------------------------
      A     "DB: AutoSPOT".StatusRx.Ndr;	//NDR ?
      JCN   CON1;	//if NO
      L     DB31.DBW 18;	//"Receive without error"
      +     1;	//increment counter
      T     DB31.DBW 18;
      L     "DB: AutoSPOT".StatusRx.Len;	//save RECEIVE-Length
      T     DB31.DBW 16;
      JU    LEAV;
// -------------------------------
// Check "Receive with error"
// -------------------------------
CON1: A     "DB: AutoSPOT".StatusRx.Error;	//ERROR ?
      JCN   CON2;	//if NO
      L     DB31.DBW 20;	//"Receive with error"
      +     1;	//increment counter
      T     DB31.DBW 20;
      L     0;
      L     "DB: AutoSPOT".StatusRx.Status;	//if STATUS <> 0
      ==I;
      JC    LEAV;
      T     DB31.DBW 22;	//save STATUS
      JU    LEAV;
// ----------------------------
// Check "Error in STATUS"
// ----------------------------
CON2: L     0;
      L     "DB: AutoSPOT".StatusRx.Status;	//if STATUS <> 0
      ==I;
      JC    LEAV;
      T     DB31.DBW 22;	//save STATUS
LEAV: CLR;
END_FUNCTION

FUNCTION "FC:Group_Change_Info" : VOID	// FC 40
VERSION : 0.1
BEGIN
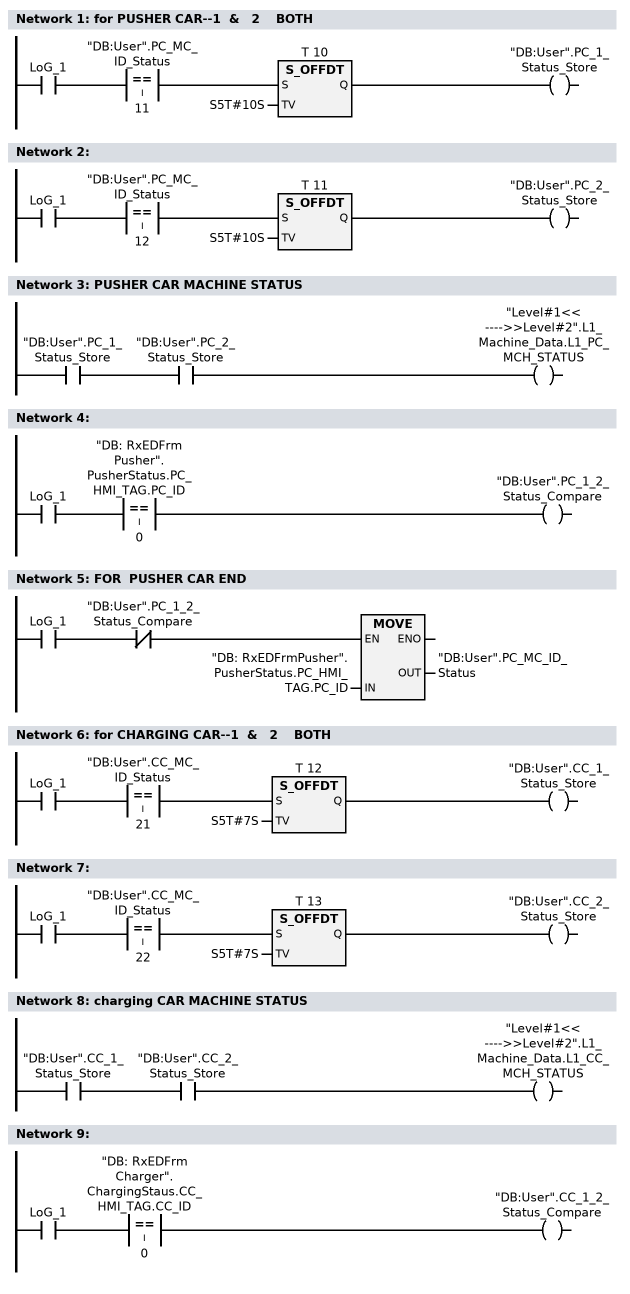
NETWORK
TITLE = for PUSHER CAR--1  &   2    BOTH
//Pusher Car Machine --1 ID Change Over Timer
      A     "LoG_1";
      A(;
      L     "DB:User".PC_MC_ID_Status;
      L     11;
      ==I;
      );
      L     S5T#10S;
      SF    T 10;
      NOP   0;
      NOP   0;
      NOP   0;
      A     T 10;
      =     "DB:User".PC_1_Status_Store;
NETWORK
TITLE =
//Pusher Car Machine --2 ID Change Over Timer
      A     "LoG_1";
      A(;
      L     "DB:User".PC_MC_ID_Status;
      L     12;
      ==I;
      );
      L     S5T#10S;
      SF    T 11;
      NOP   0;
      NOP   0;
      NOP   0;
      A     T 11;
      =     "DB:User".PC_2_Status_Store;
NETWORK
TITLE = PUSHER CAR MACHINE STATUS
//Puser Car Machine Change Over Information Go to L#2
      A     "DB:User".PC_1_Status_Store;
      A     "DB:User".PC_2_Status_Store;
      =     "Level#1<< ---->>Level#2".L1_Machine_Data.L1_PC_MCH_STATUS;
NETWORK
TITLE =
//Pusher Car 1 & 2 Bothe Nachine Compare to Zero Status
      A     "LoG_1";
      A(;
      L     "DB: RxEDFrmPusher".PusherStatus.PC_HMI_TAG.PC_ID;
      L     0;
      ==I;
      );
      =     "DB:User".PC_1_2_Status_Compare;
NETWORK
TITLE = FOR  PUSHER CAR END
//Pusher Car Macine ID Change Information
      A     "LoG_1";
      AN    "DB:User".PC_1_2_Status_Compare;
      JNB   _001;
      L     "DB: RxEDFrmPusher".PusherStatus.PC_HMI_TAG.PC_ID;
      T     "DB:User".PC_MC_ID_Status;
_001: NOP   0;
NETWORK
TITLE = for CHARGING CAR--1  &   2    BOTH
//charging Car Machine --1 ID Change Over Timer
      A     "LoG_1";
      A(;
      L     "DB:User".CC_MC_ID_Status;
      L     21;
      ==I;
      );
      L     S5T#7S;
      SF    T 12;
      NOP   0;
      NOP   0;
      NOP   0;
      A     T 12;
      =     "DB:User".CC_1_Status_Store;
NETWORK
TITLE =
//charging Car Machine --2 ID Change Over Timer
      A     "LoG_1";
      A(;
      L     "DB:User".CC_MC_ID_Status;
      L     22;
      ==I;
      );
      L     S5T#7S;
      SF    T 13;
      NOP   0;
      NOP   0;
      NOP   0;
      A     T 13;
      =     "DB:User".CC_2_Status_Store;
NETWORK
TITLE = charging CAR MACHINE STATUS
//charging Car Machine Change Over Information Go to L#2
      A     "DB:User".CC_1_Status_Store;
      A     "DB:User".CC_2_Status_Store;
      =     "Level#1<< ---->>Level#2".L1_Machine_Data.L1_CC_MCH_STATUS;
NETWORK
TITLE =
//charging Car 1 & 2 Bothe Nachine Compare to Zero Status
      A     "LoG_1";
      A(;
      L     "DB: RxEDFrmCharger".ChargingStaus.CC_HMI_TAG.CC_ID;
      L     0;
      ==I;
      );
      =     "DB:User".CC_1_2_Status_Compare;
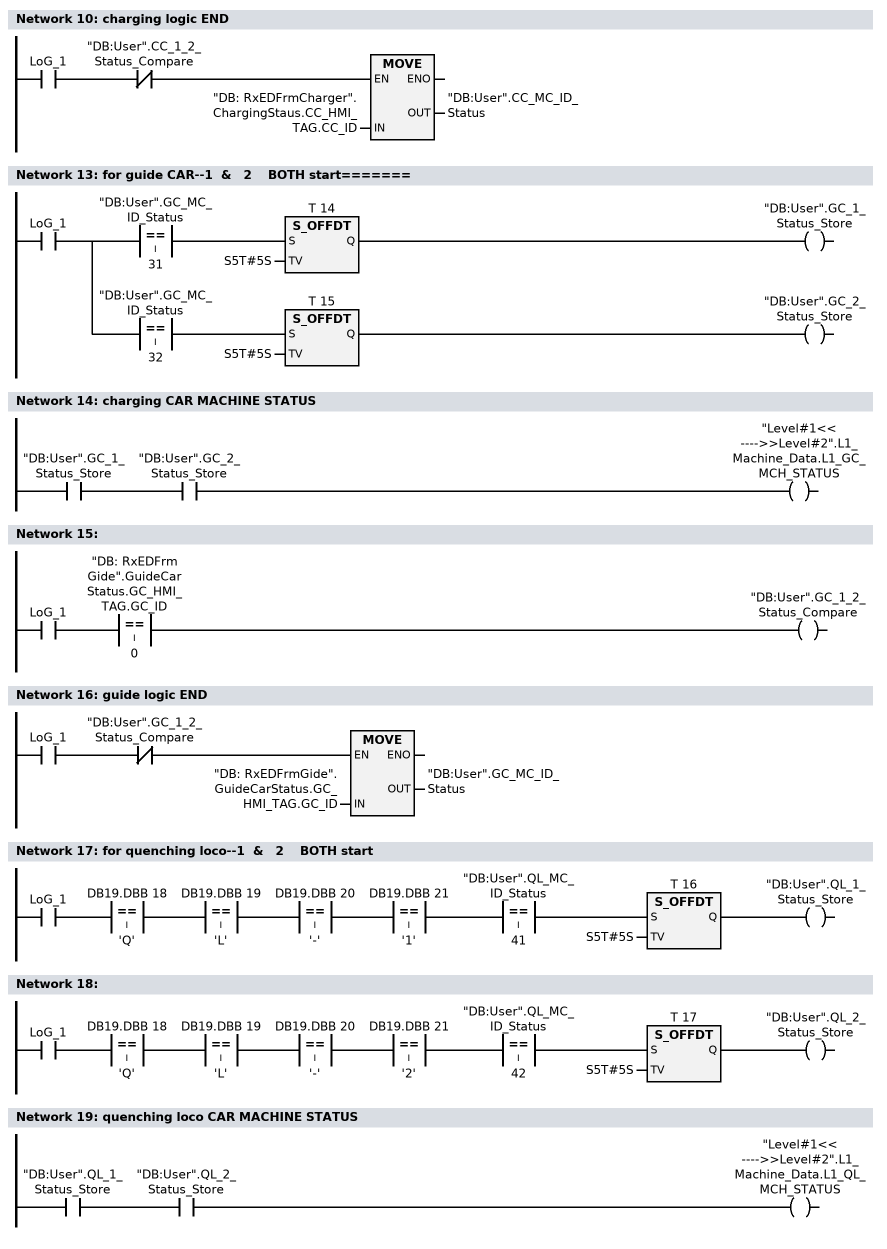
NETWORK
TITLE = charging logic END
//charging Car Macine ID Change Information
      A     "LoG_1";
      AN    "DB:User".CC_1_2_Status_Compare;
      JNB   _002;
      L     "DB: RxEDFrmCharger".ChargingStaus.CC_HMI_TAG.CC_ID;
      T     "DB:User".CC_MC_ID_Status;
_002: NOP   0;
NETWORK
TITLE = for guide CAR--1  &   2    BOTH start
//guide Car Machine --1 ID Change Over Timer
//++++++++++++++++++++++++++++++++++++++++++++++++++++++++++++++++++++++
//
//      A     "LoG_1"
//      A(    
//      L     "DB: RxEDFrmGide".GuideCarStatus.TGInfo.Description[1]
//      L     'G'
//      ==I   
//      )     
//      A(    
//      L     "DB: RxEDFrmGide".GuideCarStatus.TGInfo.Description[2]
//      L     'C'
//      ==I   
//      )     
//      A(    
//      L     "DB: RxEDFrmGide".GuideCarStatus.TGInfo.Description[3]
//      L     '-'
//      ==I   
//      )     
//      A(    
//      L     "DB: RxEDFrmGide".GuideCarStatus.TGInfo.Description[4]
//      L     '1'
//      ==I   
//      )     
//
//      A(    
//      L     "DB:User".GC_MC_ID_Status
//      L     31
//      ==I   
//      )     
//      L     S5T#5S
//      SF    T     14
//      NOP   0
//      NOP   0
//      NOP   0
//      A     T     14
//      =     "DB:User".GC_1_Status_Store
//
NETWORK
TITLE =
//guide Car Machine --2 ID Change Over Timer
//
//++++++++++++++++++++++++++++++++++++++++++++++++++++++
//      A     "LoG_1"
//      A(    
//      L     "DB: RxEDFrmGide".GuideCarStatus.TGInfo.Description[1]
//      L     'G'
//      ==I   
//      )     
//      A(    
//      L     "DB: RxEDFrmGide".GuideCarStatus.TGInfo.Description[2]
//      L     'C'
//      ==I   
//      )     
//      A(    
//      L     "DB: RxEDFrmGide".GuideCarStatus.TGInfo.Description[3]
//      L     '-'
//      ==I   
//      )     
//      A(    
//      L     "DB: RxEDFrmGide".GuideCarStatus.TGInfo.Description[4]
//      L     '2'
//      ==I   
//      )     
//      A(    
//      L     "DB:User".GC_MC_ID_Status
//      L     32
//      ==I   
//      )     
//      L     S5T#5S
//      SF    T     15
//      NOP   0
//      NOP   0
//      NOP   0
//      A     T     15
//      =     "DB:User".GC_2_Status_Store
//
NETWORK
TITLE = for guide CAR--1  &   2    BOTH start=======
      A     "LoG_1";
      =     L 0.0;
      A     L 0.0;
      A(;
      L     "DB:User".GC_MC_ID_Status;
      L     31;
      ==I;
      );
      L     S5T#5S;
      SF    T 14;
      NOP   0;
      NOP   0;
      NOP   0;
      A     T 14;
      =     "DB:User".GC_1_Status_Store;
      A     L 0.0;
      A(;
      L     "DB:User".GC_MC_ID_Status;
      L     32;
      ==I;
      );
      L     S5T#5S;
      SF    T 15;
      NOP   0;
      NOP   0;
      NOP   0;
      A     T 15;
      =     "DB:User".GC_2_Status_Store;
NETWORK
TITLE = charging CAR MACHINE STATUS
//guide Car Machine Change Over Information Go to L#2
      A     "DB:User".GC_1_Status_Store;
      A     "DB:User".GC_2_Status_Store;
      =     "Level#1<< ---->>Level#2".L1_Machine_Data.L1_GC_MCH_STATUS;
NETWORK
TITLE =
//guide Car 1 & 2 Bothe Nachine Compare to Zero Status
      A     "LoG_1";
      A(;
      L     "DB: RxEDFrmGide".GuideCarStatus.GC_HMI_TAG.GC_ID;
      L     0;
      ==I;
      );
      =     "DB:User".GC_1_2_Status_Compare;
NETWORK
TITLE = guide logic END
//guide Car Macine ID Change Information
      A     "LoG_1";
      AN    "DB:User".GC_1_2_Status_Compare;
      JNB   _003;
      L     "DB: RxEDFrmGide".GuideCarStatus.GC_HMI_TAG.GC_ID;
      T     "DB:User".GC_MC_ID_Status;
_003: NOP   0;
NETWORK
TITLE = for quenching loco--1  &   2    BOTH start
//quenching loco Machine --1 ID Change Over Timer
      A     "LoG_1";
      A(;
      L     DB19.DBB 18;
      L     'Q';
      ==I;
      );
      A(;
      L     DB19.DBB 19;
      L     'L';
      ==I;
      );
      A(;
      L     DB19.DBB 20;
      L     '-';
      ==I;
      );
      A(;
      L     DB19.DBB 21;
      L     '1';
      ==I;
      );
      A(;
      L     "DB:User".QL_MC_ID_Status;
      L     41;
      ==I;
      );
      L     S5T#5S;
      SF    T 16;
      NOP   0;
      NOP   0;
      NOP   0;
      A     T 16;
      =     "DB:User".QL_1_Status_Store;
NETWORK
TITLE =
//quenching loco Car Machine --2 ID Change Over Timer
      A     "LoG_1";
      A(;
      L     DB19.DBB 18;
      L     'Q';
      ==I;
      );
      A(;
      L     DB19.DBB 19;
      L     'L';
      ==I;
      );
      A(;
      L     DB19.DBB 20;
      L     '-';
      ==I;
      );
      A(;
      L     DB19.DBB 21;
      L     '2';
      ==I;
      );
      A(;
      L     "DB:User".QL_MC_ID_Status;
      L     42;
      ==I;
      );
      L     S5T#5S;
      SF    T 17;
      NOP   0;
      NOP   0;
      NOP   0;
      A     T 17;
      =     "DB:User".QL_2_Status_Store;
NETWORK
TITLE = quenching loco CAR MACHINE STATUS
//quenching loco Machine Change Over Information Go to L#2
      A     "DB:User".QL_1_Status_Store;
      A     "DB:User".QL_2_Status_Store;
      =     "Level#1<< ---->>Level#2".L1_Machine_Data.L1_QL_MCH_STATUS;
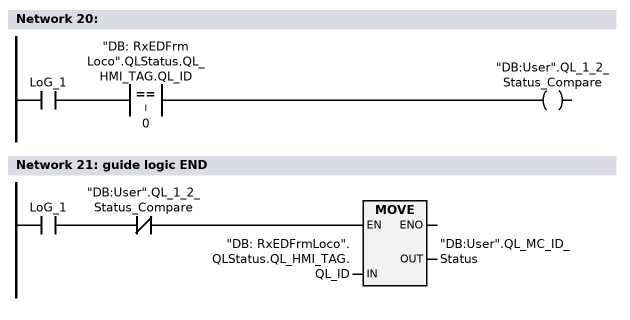
NETWORK
TITLE =
//quenching loco 1 & 2 Bothe Nachine Compare to Zero Status
      A     "LoG_1";
      A(;
      L     "DB: RxEDFrmLoco".QLStatus.QL_HMI_TAG.QL_ID;
      L     0;
      ==I;
      );
      =     "DB:User".QL_1_2_Status_Compare;
NETWORK
TITLE = guide logic END
//guide Car Macine ID Change Information
      A     "LoG_1";
      AN    "DB:User".QL_1_2_Status_Compare;
      JNB   _004;
      L     "DB: RxEDFrmLoco".QLStatus.QL_HMI_TAG.QL_ID;
      T     "DB:User".QL_MC_ID_Status;
_004: NOP   0;
END_FUNCTION

FUNCTION "FC_45_OFFLINE" : VOID	// FC 45
TITLE = moving the data to co-ordination hmi
VERSION : 0.1
VAR_TEMP
  MOV_1 : BOOL ;
  MOV_2 : BOOL ;
  MOV_3 : BOOL ;
  MOV_4 : BOOL ;
  MOV_5 : BOOL ;
  MOV_6 : BOOL ;
  MOV_7 : BOOL ;
  MOV_8 : BOOL ;
  MOV_9 : BOOL ;
  MOV_10 : BOOL ;
  MOV_11 : BOOL ;
  MOV_12 : BOOL ;
  MOV_13 : BOOL ;
  MOV_14 : BOOL ;
  MOV_15 : BOOL ;
  MOV_16 : BOOL ;
  MOV_17 : BOOL ;
  MOV_18 : BOOL ;
  MOV_19 : BOOL ;
  MOV_20 : BOOL ;
  MOV_21 : BOOL ;
  MOV_22 : BOOL ;
  MOV_23 : BOOL ;
  MOV_24 : BOOL ;
  MOV_25 : BOOL ;
  MOV_26 : BOOL ;
  MOV_27 : BOOL ;
  MOV_28 : BOOL ;
  MOV_29 : BOOL ;
  MOV_30 : BOOL ;
  MOV_31 : BOOL ;
  MOV_32 : BOOL ;
  MOV_33 : BOOL ;
  MOV_34 : BOOL ;
  MOV_35 : BOOL ;
  MOV_36 : BOOL ;
  MOV_37 : BOOL ;
  MOV_38 : BOOL ;
  MOV_39 : BOOL ;
  MOV_40 : BOOL ;
  MOV_41 : BOOL ;
  MOV_42 : BOOL ;
  MOV_43 : BOOL ;
  MOV_44 : BOOL ;
  MOV_45 : BOOL ;
  MOV_46 : BOOL ;
  MOV_47 : BOOL ;
  MOV_48 : BOOL ;
  MOV_49 : BOOL ;
  MOV_50 : BOOL ;
  MOV_51 : BOOL ;
  MOV_52 : BOOL ;
  MOV_53 : BOOL ;
  MOV_54 : BOOL ;
  MOV_55 : BOOL ;
  MOV_56 : BOOL ;
  MOV_57 : BOOL ;
  MOV_58 : BOOL ;
  MOV_59 : BOOL ;
  MOV_60 : BOOL ;
  MOV_61 : BOOL ;
  MOV_62 : BOOL ;
  MOV_63 : BOOL ;
  MOV_64 : BOOL ;
  MOV_65 : BOOL ;
  MOV_66 : BOOL ;
  MOV_67 : BOOL ;
  MOV_68 : BOOL ;
  MOV_69 : BOOL ;
  MOV_70 : BOOL ;
  MOV_71 : BOOL ;
  MOV_72 : BOOL ;
  MOV_73 : BOOL ;
  MOV_74 : BOOL ;
  MOV_75 : BOOL ;
  MOV_76 : BOOL ;
  MOV_77 : BOOL ;
  MOV_78 : BOOL ;
  MOV_79 : BOOL ;
  MOV_80 : BOOL ;
  MOV_81 : BOOL ;
  MOV_82 : BOOL ;
  MOV_83 : BOOL ;
  MOV_84 : BOOL ;
  MOV_85 : BOOL ;
  MOV_86 : BOOL ;
  MOV_87 : BOOL ;
  MOV_88 : BOOL ;
  MOV_89 : BOOL ;
  MOV_90 : BOOL ;
END_VAR
BEGIN
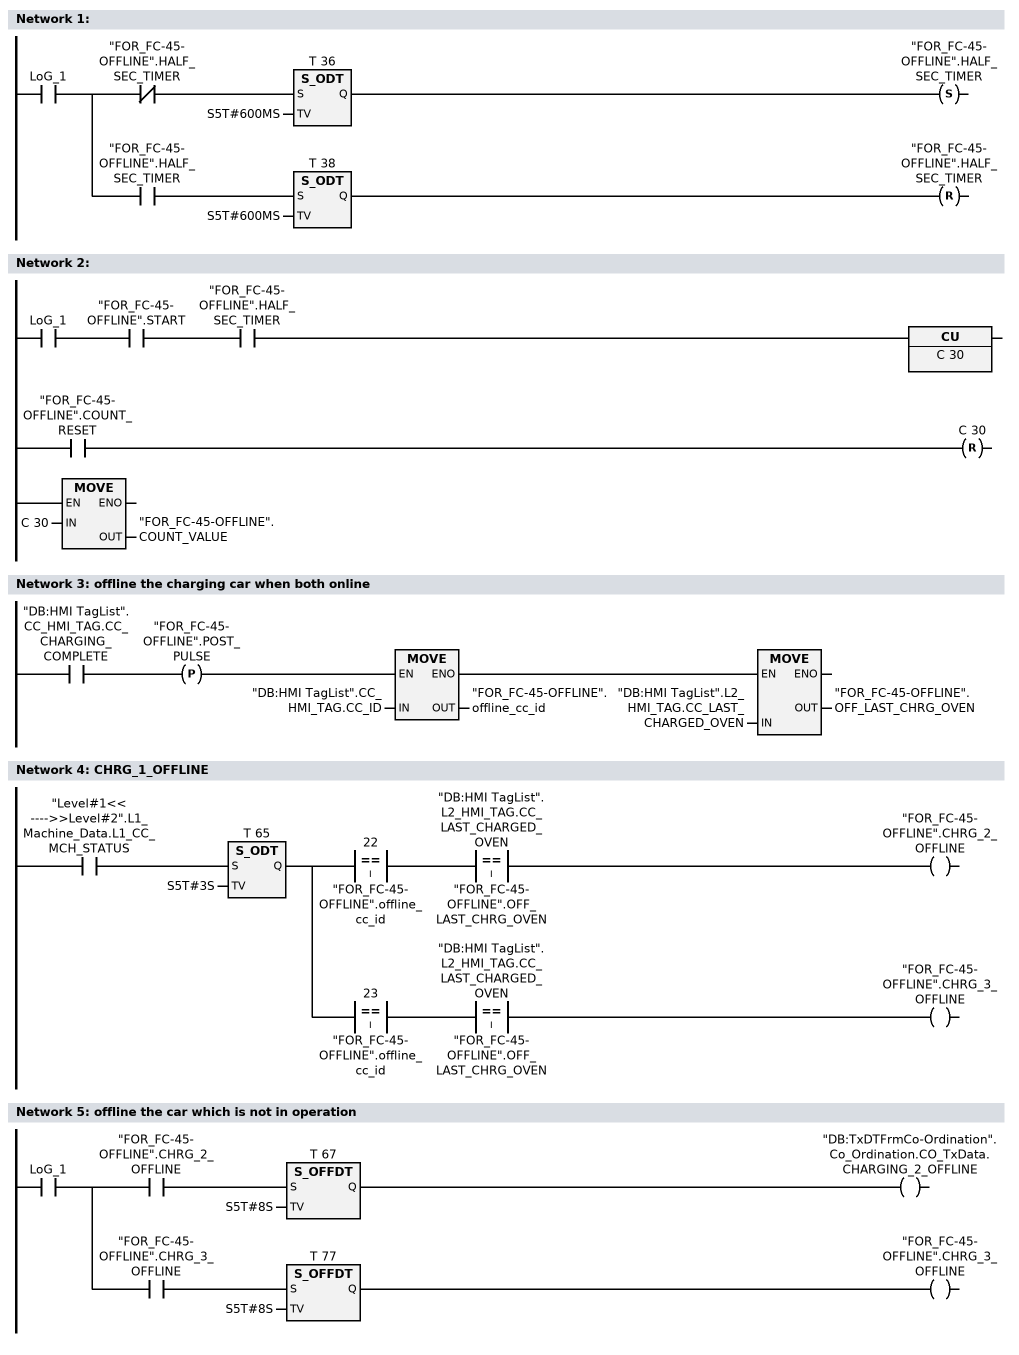
NETWORK
TITLE =
      A     "LoG_1";
      =     L 12.0;
      A     L 12.0;
      AN    "FOR_FC-45-OFFLINE".HALF_SEC_TIMER;
      L     S5T#600MS;
      SD    T 36;
      NOP   0;
      NOP   0;
      NOP   0;
      A     T 36;
      S     "FOR_FC-45-OFFLINE".HALF_SEC_TIMER;
      A     L 12.0;
      A     "FOR_FC-45-OFFLINE".HALF_SEC_TIMER;
      L     S5T#600MS;
      SD    T 38;
      NOP   0;
      NOP   0;
      NOP   0;
      A     T 38;
      R     "FOR_FC-45-OFFLINE".HALF_SEC_TIMER;
NETWORK
TITLE =
      A     "LoG_1";
      A     "FOR_FC-45-OFFLINE".START;
      A     "FOR_FC-45-OFFLINE".HALF_SEC_TIMER;
      CU    C 30;
      BLD   101;
      NOP   0;
      NOP   0;
      A     "FOR_FC-45-OFFLINE".COUNT_RESET;
      R     C 30;
      L     C 30;
      T     "FOR_FC-45-OFFLINE".COUNT_VALUE;
      NOP   0;
      NOP   0;
NETWORK
TITLE = offline the charging car when both online
//MOVE M/C ID AND CHRG OVEN
      A(;
      A     "DB:HMI TagList".CC_HMI_TAG.CC_CHARGING_COMPLETE;
      FP    "FOR_FC-45-OFFLINE".POST_PULSE;
      JNB   _001;
      L     "DB:HMI TagList".CC_HMI_TAG.CC_ID;
      T     "FOR_FC-45-OFFLINE".offline_cc_id;
      SET;
      SAVE;
      CLR;
_001: A     BR;
      );
      JNB   _002;
      L     "DB:HMI TagList".L2_HMI_TAG.CC_LAST_CHARGED_OVEN;
      T     "FOR_FC-45-OFFLINE".OFF_LAST_CHRG_OVEN;
_002: NOP   0;
NETWORK
TITLE = CHRG_1_OFFLINE
      A     "Level#1<< ---->>Level#2".L1_Machine_Data.L1_CC_MCH_STATUS;
      L     S5T#3S;
      SD    T 65;
      NOP   0;
      NOP   0;
      NOP   0;
      A     T 65;
      =     L 12.0;
      A     L 12.0;
      A(;
      L     22;
      L     "FOR_FC-45-OFFLINE".offline_cc_id;
      ==I;
      );
      A(;
      L     "DB:HMI TagList".L2_HMI_TAG.CC_LAST_CHARGED_OVEN;
      L     "FOR_FC-45-OFFLINE".OFF_LAST_CHRG_OVEN;
      ==I;
      );
      =     "FOR_FC-45-OFFLINE".CHRG_2_OFFLINE;
      A     L 12.0;
      A(;
      L     23;
      L     "FOR_FC-45-OFFLINE".offline_cc_id;
      ==I;
      );
      A(;
      L     "DB:HMI TagList".L2_HMI_TAG.CC_LAST_CHARGED_OVEN;
      L     "FOR_FC-45-OFFLINE".OFF_LAST_CHRG_OVEN;
      ==I;
      );
      =     "FOR_FC-45-OFFLINE".CHRG_3_OFFLINE;
NETWORK
TITLE = offline the car which is not in operation
      A     "LoG_1";
      =     L 12.0;
      A     L 12.0;
      A     "FOR_FC-45-OFFLINE".CHRG_2_OFFLINE;
      L     S5T#8S;
      SF    T 67;
      NOP   0;
      NOP   0;
      NOP   0;
      A     T 67;
      =     "DB:TxDTFrmCo-Ordination".Co_Ordination.CO_TxData.CHARGING_2_OFFLINE;
      A     L 12.0;
      A     "FOR_FC-45-OFFLINE".CHRG_3_OFFLINE;
      L     S5T#8S;
      SF    T 77;
      NOP   0;
      NOP   0;
      NOP   0;
      A     T 77;
      =     "FOR_FC-45-OFFLINE".CHRG_3_OFFLINE;
END_FUNCTION

DATA_BLOCK "DB:RxDTFrmPushCurrent"	// DB 15
VERSION : 0.1
  STRUCT
   Pusher_Ram : STRUCT
    TGInfo : STRUCT
     Header : CHAR  := '!';	//Telegram Header
     SenderID : INT ;	//Sender's ID (Unique Machine/Equipment ID)
     Recipients : INT ;	//Recipients (1 Bit for Each Recipient) - Ignored
     TGramID : INT ;	//Unique Telegram ID
     TXMnNo : BYTE ;	//Transmission Number
     LenMsg : INT ;	//Length In Bytes
     CRCAdd : WORD ;	//Additive CRC
     RxMnNo : WORD ;
     Description : STRING  [4 ];
    END_STRUCT ;
    PC_Current : STRUCT
     RamCurrent : ARRAY  [1 .. 90 ] OF INT ;
    END_STRUCT ;
   END_STRUCT ;
  END_STRUCT ;	
BEGIN
   Pusher_Ram.TGInfo.Header := '!';
END_DATA_BLOCK

DATA_BLOCK "DB:RxDTFrmLavelleCurrent"	// DB 16
VERSION : 0.1
  STRUCT
   Pusher_Laveller : STRUCT
    TGInfo : STRUCT
     Header : CHAR  := '!';	//Telegram Header
     SenderID : INT ;	//Sender's ID (Unique Machine/Equipment ID)
     Recipients : INT ;	//Recipients (1 Bit for Each Recipient) - Ignored
     TGramID : INT ;	//Unique Telegram ID
     TXMnNo : BYTE ;	//Transmission Number
     LenMsg : INT ;	//Length In Bytes
     CRCAdd : WORD ;	//Additive CRC
     RxMnNo : WORD ;
     Description : STRING  [4 ];
    END_STRUCT ;
    PC_Laveller_Current : STRUCT
     LavellerCurrent : ARRAY  [1 .. 90 ] OF INT ;
    END_STRUCT ;
   END_STRUCT ;
  END_STRUCT ;	
BEGIN
   Pusher_Laveller.TGInfo.Header := '!';
END_DATA_BLOCK

DATA_BLOCK "DB: RxEDFrmCharger"	// DB 17
VERSION : 0.1
  STRUCT
   ChargingStaus : STRUCT
    TGInfo : STRUCT
     Header : CHAR  := '!';	//Telegram Header
     SenderID : INT ;	//Sender's ID (Unique Machine/Equipment ID)
     Recipients : INT ;	//Recipients (1 Bit for Each Recipient) - Ignored
     TGramID : INT ;	//Unique Telegram ID
     TXMnNo : BYTE ;	//Transmission Number
     LenMsg : INT ;	//Length In Bytes
     CRCAdd : WORD ;	//Additive CRC
     RxMnNo : WORD ;
     Description : STRING  [4 ];
    END_STRUCT ;
    CC_HMI_TAG : STRUCT
     CC_RF_Communicating : BOOL ;	//Charging car RF communication Helthy
     CC_Enc_STATUS : BOOL ;	//Encoder Status for CC
     CC_RF_STATUS : BOOL ;	//RF Modem Status for CC
     CC_AutoSpot_STATUS : BOOL ;	//AutoSPOT  Status for CC
     LEVLLING_STOP : BOOL ;	//Field Devices (ENC, plc, AutoSPOT, & RF) Status Combined
     CC_MCH_STATUS : BOOL ;	//Machine Health & Operation Status for CC
     CC_ALIGN_STATUS : BOOL ;	//Machine Align Status Against Target Oven for CC
     CC_PERM : BOOL ;	//Manual confirmation (leveling to  start)
     LEVLLING_START : BOOL ;	//LEVLLEING in progress
     CC_GRP_STATUS : INT ;	//Indicate Whether The Machine Is In The Group Or Out Of Group
     CC_ID : INT ;	//Machine ID for CC
     CC_OVEN_ID_ACT : INT ;	//Oven ID of Present Location for CC
     CC_CHARGING_START : BOOL ;	//CHARGING START
     CC_CHARGING_COMPLETE : BOOL ;	//CHARGING COMPLETE
    END_STRUCT ;
   END_STRUCT ;
  END_STRUCT ;	
BEGIN
   ChargingStaus.TGInfo.Header := '!';
END_DATA_BLOCK

DATA_BLOCK "DB: RxEDFrmGide"	// DB 18
VERSION : 0.1
  STRUCT
   GuideCarStatus : STRUCT
    TGInfo : STRUCT
     Header : CHAR  := '!';	//Telegram Header
     SenderID : INT ;	//Sender's ID (Unique Machine/Equipment ID)
     Recipients : INT ;	//Recipients (1 Bit for Each Recipient) - Ignored
     TGramID : INT ;	//Unique Telegram ID
     TXMnNo : BYTE ;	//Transmission Number
     LenMsg : INT ;	//Length In Bytes
     CRCAdd : WORD ;	//Additive CRC
     RxMnNo : WORD ;
     Description : STRING  [4 ];
    END_STRUCT ;
    GC_HMI_TAG : STRUCT
     GC_RF_Communicating : BOOL ;	//Charging car RF communication Helthy
     GC_Enc_STATUS : BOOL ;	//Encoder Status for GC
     GC_RF_STATUS : BOOL ;	//RF Modem Status for GC
     GC_AutoSpot_STATUS : BOOL ;	//AutoSPOT  Status for GC
     GC_FLD_STATUS : BOOL ;	//Field Devices (ENC, plc, AutoSPOT, & RF) Status Combined
     GC_MCH_STATUS : BOOL ;	//Machine Health & Operation Status for GC
     GC_ALIGN_STATUS : BOOL ;	//Machine Align Status Against Target Oven for GC
     GC_PERM : BOOL ;	//Manual confirmation
     Spare_0 : BOOL ;
     GC_GRP_STATUS : INT ;	//Indicate Whether The Machine Is In The Group Or Out Of Group
     GC_ID : INT ;	//Machine ID for GC
     GC_OVEN_ID_ACT : INT ;	//Oven ID of Present Location for GC
    END_STRUCT ;
   END_STRUCT ;
  END_STRUCT ;	
BEGIN
   GuideCarStatus.TGInfo.Header := '!';
END_DATA_BLOCK

DATA_BLOCK "DB: RxEDFrmLoco"	// DB 19
VERSION : 0.1
  STRUCT
   QLStatus : STRUCT
    TGInfo : STRUCT
     Header : CHAR  := '!';	//Telegram Header
     SenderID : INT ;	//Sender's ID (Unique Machine/Equipment ID)
     Recipients : INT ;	//Recipients (1 Bit for Each Recipient) - Ignored
     TGramID : INT ;	//Unique Telegram ID
     TXMnNo : BYTE ;	//Transmission Number
     LenMsg : INT ;	//Length In Bytes
     CRCAdd : WORD ;	//Additive CRC
     RxMnNo : WORD ;
     Description : STRING  [4 ];
    END_STRUCT ;
    QL_HMI_TAG : STRUCT
     QL_RF_Communicating : BOOL ;	//RF communication OK
     QL_Enc_STATUS : BOOL ;	//Encoder Status for QL
     QL_RF_STATUS : BOOL ;	//RF Modem Status for QL
     QL_AutoSpot_STATUS : BOOL ;	//AutoSPOT  Status for QL
     QL_FLD_STATUS : BOOL ;	//Field Devices (ENC, plc, AutoSPOT, & RF) Status Combined
     QL_MCH_STATUS : BOOL ;	//Machine Health & Operation Status for QL
     QL_ALIGN_STATUS : BOOL ;	// (1=Aligned)
     QL_PERM : BOOL ;	//Manual confirmation (QL is ready to receive coke)
     Spare0 : BOOL ;	//Current LT Mode (1-Auto/0-Manual)
     Spare1 : BOOL ;	//Request for moving battery#1
     Spare2 : BOOL ;	//Request for moving battery#2
     QL_GRP_STATUS : INT ;	//Indicate Whether The Machine Is In The Group Or Out Of Group(1-bat#1,2-bat#2,)
     QL_ID : INT ;	//Machine ID for QL
     QL_OVEN_ID_ACT : INT ;	//Oven ID of Present Location for QL
     QL_POS : DINT ;	//Location of QL During Loco Synchronization
    END_STRUCT ;
   END_STRUCT ;
  END_STRUCT ;	
BEGIN
   QLStatus.TGInfo.Header := '!';
END_DATA_BLOCK

DATA_BLOCK "DB: RxEDFrmPusher"	// DB 20
VERSION : 0.1
  STRUCT
   PusherStatus : STRUCT
    TGInfo : STRUCT
     Header : CHAR  := '!';	//Telegram Header
     SenderID : INT ;	//Sender's ID (Unique Machine/Equipment ID)
     Recipients : INT ;	//Recipients (1 Bit for Each Recipient) - Ignored
     TGramID : INT ;	//Unique Telegram ID
     TXMnNo : BYTE ;	//Transmission Number
     LenMsg : INT ;	//Length In Bytes
     CRCAdd : WORD ;	//Additive CRC
     RxMnNo : WORD ;
     Description : STRING  [4 ];
    END_STRUCT ;
    PC_HMI_TAG : STRUCT
     PC_RF_Communicating : BOOL ;	//Pusher car RF communication Helthy
     PC_Enc_STATUS : BOOL ;	//Encoder Status for PC
     PC_RF_STATUS : BOOL ;	//RF Modem Status for PC
     PC_AutoSpot_STATUS : BOOL ;	//AutoSPOT  Status for PC
     Push_complite : BOOL ;
     PC_MCH_STATUS : BOOL ;	//Machine Health & Operation Status for PC
     PC_ALIGN_STATUS : BOOL ;	//Machine Align Status Against Target Oven for PC
     PC_PERM : BOOL ;	//Manual confirmation (leveling to  start)
     LEVLLING_PERM : BOOL ;	//LEVLLEING in progress
     Spare00 : BOOL ;
     Spare01 : BOOL ;
     Push_Start : BOOL ;	//Pushing Started
     Spare03 : BOOL ;
     Spare04 : BOOL ;
     Spare05 : BOOL ;
     Spare06 : BOOL ;
     PC_GRP_STATUS : INT ;	//Indicate Whether The Machine Is In The Group Or Out Of Group
     PC_ID : INT ;	//Machine ID for PC
     PC_OVEN_ID_ACT : INT ;	//Oven ID of Present Location for PC
     PC_RAM_Position : DINT ;	//PUSHER RAM POSITION
     PC_PUSHING_CURRENT : INT ;	//PUSHER RAM CURRENT
     PC_LEVELLING_CURRENT : INT ;	//PUSHER LEVELLER CURRENT
    END_STRUCT ;
   END_STRUCT ;
  END_STRUCT ;	
BEGIN
   PusherStatus.TGInfo.Header := '!';
   PusherStatus.PC_HMI_TAG.Push_complite := TRUE;
END_DATA_BLOCK

DATA_BLOCK "DB:TxDTFrmCo-Ordination"	// DB 21
VERSION : 0.1
  STRUCT
   Co_Ordination : STRUCT
    TGInfo : STRUCT
     Header : CHAR  := '!';	//Telegram Header
     SenderID : INT  := 1;	//Sender's ID (Unique Machine/Equipment ID)
     Recipients : INT ;	//Recipients (1 Bit for Each Recipient) - Ignored
     TGramID : INT  := 21;	//Unique Telegram ID
     TXMnNo : BYTE  := B#16#10;	//Transmission Number
     LenMsg : INT  := 167;	//Length In Bytes
     CRCAdd : WORD ;	//Additive CRC
     RxMnNo : WORD ;
     Description : STRING  [4 ] := 'CO-1';
    END_STRUCT ;
    CO_TxData : STRUCT
     Co_Communicating : BOOL ;
     SCH_1_OVEN_ID : INT ;	//SCH_1_OVEN_ID
     SCH_1_ACT_MOMENT : STRING  [17 ];	//SCH_1_ACT_MOMENT
     SCH_1_SERIAL_NO : INT ;	//SCH_1_SERIAL_NO
     SCH_1_ACTION : STRING  [1 ] := ' ';	//SCH_1_ACTION ( 'P'=PUSHING 'C'=CHARGING)
     SCH_2_OVEN_ID : INT ;	//SCH_2_OVEN_ID
     SCH_2_ACT_MOMENT : STRING  [17 ];	//SCH_2_ACT_MOMENT
     SCH_2_SERIAL_NO : INT ;	//SCH_2_SERIAL_NO
     SCH_2_ACTION : STRING  [1 ] := ' ';	//SCH_2_ACTION ( 'P'=PUSHING 'C'=CHARGING)
     SCH_3_OVEN_ID : INT ;	//SCH_3_OVEN_ID
     SCH_3_ACT_MOMENT : STRING  [17 ];	//SCH_3_ACT_MOMENT
     SCH_3_SERIAL_NO : INT ;	//SCH_3_SERIAL_NO
     SCH_3_ACTION : STRING  [1 ] := ' ';	//SCH_3_ACTION ( 'P'=PUSHING 'C'=CHARGING)
     SCH_4_OVEN_ID : INT ;	//SCH_4_OVEN_ID
     SCH_4_ACT_MOMENT : STRING  [17 ];	//SCH_4_ACT_MOMENT
     SCH_4_SERIAL_NO : INT ;	//SCH_4_SERIAL_NO
     SCH_4_ACTION : STRING  [1 ] := ' ';	//SCH_4_ACTION ( 'P'=PUSHING 'C'=CHARGING)
     SCH_5_OVEN_ID : INT ;	//SCH_5_OVEN_ID
     SCH_5_ACT_MOMENT : STRING  [17 ];	//SCH_5_ACT_MOMENT
     SCH_5_SERIAL_NO : INT ;	//SCH_5_SERIAL_NO
     SCH_5_ACTION : STRING  [1 ] := ' ';	//SCH_5_ACTION ( 'P'=PUSHING 'C'=CHARGING)
     SPARE : INT ;	//OFFLINE_WHEN_BOTH_CHARGING_CAR_ONLINE
     CHARGING_1_OFFLINE : BOOL ;	//CHARGING_1_OFFLINE
     CHARGING_2_OFFLINE : BOOL ;	//CHARGING_2_OFFLINE
     CHARGING_3_OFFLINE : BOOL ;	//CHARGING_3_OFFLINE
     SPARE11 : BOOL ;
     SPARE12 : BOOL ;
     SPARE13 : BOOL ;
     SPARE14 : BOOL ;
     SPARE15 : BOOL ;
    END_STRUCT ;
   END_STRUCT ;
  END_STRUCT ;	
BEGIN
   Co_Ordination.TGInfo.Header := '!';
   Co_Ordination.TGInfo.SenderID := 1;
   Co_Ordination.TGInfo.TGramID := 21;
   Co_Ordination.TGInfo.TXMnNo := B#16#10;
   Co_Ordination.TGInfo.LenMsg := 167;
   Co_Ordination.TGInfo.Description := 'CO-1';
   Co_Ordination.CO_TxData.SCH_1_ACTION := ' ';
   Co_Ordination.CO_TxData.SCH_2_ACTION := ' ';
   Co_Ordination.CO_TxData.SCH_3_ACTION := ' ';
   Co_Ordination.CO_TxData.SCH_4_ACTION := ' ';
   Co_Ordination.CO_TxData.SCH_5_SERIAL_NO := 4;
   Co_Ordination.CO_TxData.SCH_5_ACTION := ' ';
END_DATA_BLOCK

DATA_BLOCK "Level#1<< ---->>Level#2"	// DB 23
VERSION : 0.1
  STRUCT
   L1_Machine_Data : STRUCT
    L1_PC_PUSH_COMPLETE : BOOL ;	//PUSHING COMPLETE
    L1_PC_MCH_STATUS : BOOL ;	//PUSHER CAR MACHINE STATUS
    L1_CC_MCH_STATUS : BOOL ;	//CHARGING CAR MACHINE STATUS
    L1_GC_MCH_STATUS : BOOL ;	//GUIDE CAR MACHINE STATUS
    L1_QL_MCH_STATUS : BOOL ;	//QUENCHING LOCO CAR MACHINE STATUS
    L1_PC_PUSH_START : BOOL ;	//PUSHING STARTED
    SPARE0_6 : BOOL ;
    L1_CC_CHARG_START : BOOL ;	//CHARGING STARTED
    L1_CC_CHARG_COMPLETE : BOOL ;	//CHARGING COMPLETE
    L1_SCH_SENT : BOOL ;	//SCHEDULE SENT UPDATE BIT
    L1_BOTH_PC_ONLINE : BOOL ;
    L1_BOTH_CC_ONLINE : BOOL ;
    L1_BOTH_GC_ONLINE : BOOL ;
    L1_BOTH_QL_ONLINE : BOOL ;
    SPARE1_6 : BOOL ;
    SPARE1_7 : BOOL ;
    L1_PC_MCHID : INT ;	//MACHINE NUMBER OF THE PUSHER CAR
    L1_PC_POSID : INT ;	//OVEN NUMBER AS THE MACHINE PASSES BY THE OVEN
    L1_PC_ACT_POSID : INT ;	//OVEN NUMBER WHERE THE MACHINE IS PUSHING
    L1_PC_GRP_STATUS : INT ;
    SPARE10_0 : INT ;
    L1_CC_MCHID : INT ;	//MACHINE NUMBER OF THE CHARGING CAR
    L1_CC_POSID : INT ;	//OVEN NUMBER AS THE MACHINE PASSES BY THE OVEN
    LI_CC_ACT_POSID : INT ;	//OVEN NUMBER WHERE THE MACHINE IS CHARGING
    L1_CC_GRP_STATUS : INT ;
    SPARE20_0 : INT ;
    L1_GC_MCHID : INT ;	//MACHINE NUMBER OF THE GUIDE CAR
    L1_GC_POSID : INT ;	//OVEN NUMBER AS THE MACHINE PASSES BY THE OVEN
    L1_GC_ACT_POSID : INT ;	//OVEN NUMBER AS THE MACHINE IS FORWARDING THE DOOR EXTRACTOR
    L1_GC_GRP_STATUS : INT ;
    SPARE30_0 : INT ;
    L1_QL_MCHID : INT ;	//MACHINE NUMBER OF THE QUENCHING LOCO CAR
    L1_QL_POSID : INT ;	//OVEN NUMBER AS THE MACHINE PASSES BY THE OVEN
    L1_QL_ACT_POSID : INT ;	//OVEN NUMBER WHERE THE MACHINE IS STANDING TO RECIEVE COKE
    L1_QL_GRP_STATUS : INT ;
    SPARE40_0 : INT ;
    L1_PC_RAM_POSITION : DINT ;	//PUSHING CAR RAM POSITION
    STAT_0 : REAL ;
   END_STRUCT ;
   L2_Servar_Data : STRUCT
    L1_SCH_1_OVEN_ID : INT ;
    L1_SCH_1_ACT_MOMENT : STRING  [17 ];
    L1_SCH_1_SERIAL_NO : INT ;
    L1_SCH_1_ACTION : STRING  [1 ];
    L1_SCH_2_OVEN_ID : INT ;
    L1_SCH_2_ACT_MOMENT : STRING  [17 ];
    L1_SCH_2_SERIAL_NO : INT ;
    L1_SCH_2_ACTION : STRING  [1 ];
    L1_SCH_3_OVEN_ID : INT ;
    L1_SCH_3_ACT_MOMENT : STRING  [17 ];
    L1_SCH_3_SERIAL_NO : INT ;
    L1_SCH_3_ACTION : STRING  [1 ];
    L1_SCH_4_OVEN_ID : INT ;
    L1_SCH_4_ACT_MOMENT : STRING  [17 ];
    L1_SCH_4_SERIAL_NO : INT ;
    L1_SCH_4_ACTION : STRING  [1 ];
    L1_SCH_5_OVEN_ID : INT ;
    L1_SCH_5_ACT_MOMENT : STRING  [17 ];
    L1_SCH_5_SERIAL_NO : INT ;
    L1_SCH_5_ACTION : STRING  [1 ];
   END_STRUCT ;
   Sata_1 : BOOL ;
   Sata_2 : BOOL ;
   Sata_3 : BOOL ;
   Sata_4 : BOOL ;
   Sata_5 : BOOL ;
   Sata_6 : BOOL ;
   Sata_7 : BOOL ;
   Sata_8 : BOOL ;
   L1_PusherCar_Data : STRUCT
    RAM_CURRENT : ARRAY  [1 .. 90 ] OF //PUSHER CAR RAM CURRENT
    INT ;
    LEVELLER_CURRENT : ARRAY  [1 .. 90 ] OF //PUSHER CAR LEVELLER CURRENT
    INT ;
   END_STRUCT ;
  END_STRUCT ;	
BEGIN
   L2_Servar_Data.L1_SCH_1_SERIAL_NO := 1;
END_DATA_BLOCK

DATA_BLOCK "DB:Data_ReciveBuffer"	// DB 29
VERSION : 0.1
  STRUCT
   REcivedBuffer_Freq : ARRAY  [1 .. 500 ] OF //RF Recived Buffer
   BYTE ;
  END_STRUCT ;	
BEGIN
END_DATA_BLOCK

DATA_BLOCK "DB: AutoSPOT"	// DB 31
VERSION : 0.1
  STRUCT
   OPs : STRUCT
    OvenID : INT ;	//Oven Number Machine Is Aligned At.
    Aligned : BOOL ;	//True = Machine Is Aligned At Oven=OvenID Else Not
    S9Aligned : BOOL ;	//True = If S9/Left Marker Is Blocked
    S10Aligned : BOOL ;	//True = If S10/Right Marker Is Blocked
    McInWrongBatt : BOOL ;	//True If Machine Movement In Wrong Battery
    UnitID : INT ;	//UnitID Of Connected AutoSPOT H/w
    LinkFail : BOOL ;	//True = If Communication Error, Bad Data Etc.
   END_STRUCT ;
   StatusRx : STRUCT
    Ndr : BOOL ;	//Read CP (FB7 Block) Ndr Values
    Error : BOOL ;	//Read CP (FB7 Block) Error Values
    Len : INT ;	//Read CP (FB7 Block) Len Values
    Status : WORD ;	//Read CP (FB7 Block) Status Values
    PktRxED : BOOL ;	//=True whenever a packet is recieved.
    PktVerified : BOOL ;	//=True whenever a packet is verified.
    LinkFail : BOOL ;	//=True whenever there is no data from AutoSPOT for long
    IsAbsolutePos : BOOL ;	//=True If Marker Plate Is for Absolute Locations Like Quenching Tower Etc.
   END_STRUCT ;
   Spares : STRUCT
    DUMMY : ARRAY  [1 .. 34 ] OF BYTE ;
   END_STRUCT ;
   TGram : STRUCT
    HDR : BYTE ;	//=AA Hex
    TGID : BYTE ;	//=01 (Signature, Not Aligned), =02 Information (Algined)
    MarVal : BYTE ;	//XXXX-XXS10S9(give d marker alues 0,1,2,3)
    PltAdr : BYTE ;	//S8S7S6S5-S4S3S2S1(give d number read by auto spot)
    Free1 : BYTE ;	//=55 Hex
    Free2 : BYTE ;	//=55 Hex
    CRCHigh : BYTE ;
    CRCLow : BYTE ;
    UnitID : BYTE ;
    FTR1 : BYTE ;	//=20 Hex
    FTR2 : BYTE ;	//=CR
    FTR3 : BYTE ;	//=LF
   END_STRUCT ;
   EXTRA_BUFFER : ARRAY  [1 .. 128 ] OF BYTE ;
  END_STRUCT ;	
BEGIN
   TGram.TGID := B#16#2;
   TGram.PltAdr := B#16#1F;
END_DATA_BLOCK

DATA_BLOCK "DB: RFModem Freq"	// DB 32
VERSION : 0.1
  STRUCT
   TGram_SelNSaveBat1Freq : STRUCT
    VAR1 : CHAR  := 'S';
    VAR2 : CHAR  := 'L';
    VAR3 : CHAR  := '&';
    VAR4 : CHAR  := 'F';
    VAR5 : CHAR  := '=';
    FREQ1 : CHAR  := '4';
    FREQ2 : CHAR  := '3';
    FREQ3 : CHAR  := '7';
    FREQ4 : CHAR  := '.';
    FREQ5 : CHAR  := '1';
   END_STRUCT ;
   TGram_SelNSaveBat2Freq : STRUCT 	//Frequency F2=436.1Hz NOT for Battery#1
    VAR1 : CHAR  := 'S';	//This Set Of Data not required for Battery#1 (CC-1;PC-1;GC-1;QL-1)
    VAR2 : CHAR  := 'L';
    VAR3 : CHAR  := '&';
    VAR4 : CHAR  := 'F';
    VAR5 : CHAR  := '=';
    FREQ1 : CHAR  := '4';
    FREQ2 : CHAR  := '3';
    FREQ3 : CHAR  := '7';
    FREQ4 : CHAR  := '.';
    FREQ5 : CHAR  := '2';
   END_STRUCT ;
   TGram_SelNSaveOffLine : STRUCT
    VAR1 : CHAR  := 'S';
    VAR2 : CHAR  := 'L';
    VAR3 : CHAR  := '&';
    VAR4 : CHAR  := 'F';
    VAR5 : CHAR  := '=';
    FREQ1 : CHAR  := '4';
    FREQ2 : CHAR  := '3';
    FREQ3 : CHAR  := '7';
    FREQ4 : CHAR  := '.';
    FREQ5 : CHAR  := '8';
   END_STRUCT ;
   TGram_SaveMdmSettings : STRUCT
    VAR1 : CHAR  := 'S';
    VAR2 : CHAR  := 'L';
    VAR3 : CHAR  := '*';
    VAR4 : CHAR  := '*';
    VAR5 : CHAR  := '>';
   END_STRUCT ;
   TGram_MachineGrouping : STRUCT
    Header : STRUCT
     MsgLen : INT ;	//Length of Message
     MsgID : BYTE ;
    END_STRUCT ;
    MachineName : CHAR ;
    MachineNo : INT ;
    MachineFrequency : INT ;
    BatteryNo : INT  := 2;
   END_STRUCT ;
  END_STRUCT ;	
BEGIN
   TGram_SelNSaveBat1Freq.VAR1 := 'S';
   TGram_SelNSaveBat1Freq.VAR2 := 'L';
   TGram_SelNSaveBat1Freq.VAR3 := '&';
   TGram_SelNSaveBat1Freq.VAR4 := 'F';
   TGram_SelNSaveBat1Freq.VAR5 := '=';
   TGram_SelNSaveBat1Freq.FREQ1 := '4';
   TGram_SelNSaveBat1Freq.FREQ2 := '3';
   TGram_SelNSaveBat1Freq.FREQ3 := '7';
   TGram_SelNSaveBat1Freq.FREQ4 := '.';
   TGram_SelNSaveBat1Freq.FREQ5 := '1';
   TGram_SelNSaveBat2Freq.VAR1 := 'S';
   TGram_SelNSaveBat2Freq.VAR2 := 'L';
   TGram_SelNSaveBat2Freq.VAR3 := '&';
   TGram_SelNSaveBat2Freq.VAR4 := 'F';
   TGram_SelNSaveBat2Freq.VAR5 := '=';
   TGram_SelNSaveBat2Freq.FREQ1 := '4';
   TGram_SelNSaveBat2Freq.FREQ2 := '3';
   TGram_SelNSaveBat2Freq.FREQ3 := '7';
   TGram_SelNSaveBat2Freq.FREQ4 := '.';
   TGram_SelNSaveBat2Freq.FREQ5 := '2';
   TGram_SelNSaveOffLine.VAR1 := 'S';
   TGram_SelNSaveOffLine.VAR2 := 'L';
   TGram_SelNSaveOffLine.VAR3 := '&';
   TGram_SelNSaveOffLine.VAR4 := 'F';
   TGram_SelNSaveOffLine.VAR5 := '=';
   TGram_SelNSaveOffLine.FREQ1 := '4';
   TGram_SelNSaveOffLine.FREQ2 := '3';
   TGram_SelNSaveOffLine.FREQ3 := '7';
   TGram_SelNSaveOffLine.FREQ4 := '.';
   TGram_SelNSaveOffLine.FREQ5 := '8';
   TGram_SaveMdmSettings.VAR1 := 'S';
   TGram_SaveMdmSettings.VAR2 := 'L';
   TGram_SaveMdmSettings.VAR3 := '*';
   TGram_SaveMdmSettings.VAR4 := '*';
   TGram_SaveMdmSettings.VAR5 := '>';
   TGram_MachineGrouping.MachineName := ' ';
   TGram_MachineGrouping.BatteryNo := 2;
END_DATA_BLOCK

DATA_BLOCK "DB:HMI TagList"	// DB 35
VERSION : 0.1
  STRUCT
   All_Macmine_HMI_TAG : STRUCT
    MODE_SEL_REQ : BOOL ;	//MODE SELECTION REQUEST(1-AUTO/0-MANUAL)
    CURR_LT_MODE : BOOL ;	//CURR_LT_MODE(1-AUTO/0-MANUAL)
    SELECT_BATTERY_1 : BOOL ;	//SELECT_BATTERY#1 SELECTION REQUEST
    SELECT_BATTERY_2 : BOOL ;	//SELECT_BATTERY#2 SELECTION REQUEST
    BATTERY_SEL_OFFLINE : BOOL ;	//MACHINE OFFLINE SELECTION REQUEST
    LT_START : BOOL ;	//LONG TRAVEL AUTO POSITIONING REQUEST
    JOG_R : BOOL ;	//LONG TRAVEL JOG-RIGHT REQUEST
    JOG_F : BOOL ;	//LONG TRAVEL JOG-LEFT REQUEST
    FIRING_START : BOOL ;	//MOVE TO START OF FIRING LOCATION REQUEST
    FIRING_COMPLETE : BOOL ;	//MOVE TO END OF FIRING LOCATION REQUEST
    DOOR_DELIVERY : BOOL ;	//MOVE TO DOOR DELIVERY LOCATION REQUEST
    DOOR_COLLECTION : BOOL ;	//MOVE TO DOOR COLLECTION LOCATION REQUEST
    MANUAL_SCHEDULE : BOOL ;	//SCHEDULING REQUEST(0-LEVEL-11, 1-PUSHER)
    MACHINE_INTERLOCK : BOOL ;	//MACHINE INTERLOCK DISPLAY REQUEST(OPEN POP UP)
    PUSH_REQUEST : BOOL ;	//PUSHING PERMISSIVE REQUEST(BUTTON)
    LEVELG_REQUEST : BOOL ;	//LEVELLING PERMISSIVE REQUEST(BUTTON)
    STOP_PUSHING : BOOL ;	//STOP PUSHING FOR PUSHER CAR
    GC_ReadyFor_Coke : BOOL ;
    QL_ReadyFor_Coke : BOOL ;
    PushingPermission : BOOL ;
    PC_LT_Permission : BOOL ;
    MC_LFT_ALING : BOOL ;
    MC_RIGHT_ALING : BOOL ;
    MC_AILNG : BOOL ;
    Travelling_Distance_MM : REAL ;
    Actual_Speed : REAL ;
    CC_Communication_Err : BOOL ;
    GC_Communication_Err : BOOL ;
    QL_Communication_Err : BOOL ;
    PC_Communication_Err : BOOL ;
    PC_Aliange_Bypass : BOOL ;
    Frequency_SeT : BOOL ;
    PC_PEMISSION_ACCEPT : BOOL ;
    PUSHING_COMPLETE : BOOL ;
    SPAR_TAG : ARRAY  [0 .. 3 ] OF INT ;
   END_STRUCT ;
   PC_HMI_TAG : STRUCT
    PP_RF_Communicating : BOOL ;	//RF communication OK
    PC_Enc_STATUS : BOOL ;	//Encoder Status for PC
    PC_RF_STATUS : BOOL ;	//RF Modem Status for PC
    PC_AutoSpot_STATUS : BOOL ;	//AutoSPOT  Status for PC
    PC_FLD_STATUS : BOOL ;	//Field Devices (ENC, plc, AutoSPOT, & RF) Status Combined
    PC_MCH_STATUS : BOOL ;	//Machine Health & Operation Status for PC
    PC_ALIGN_STATUS : BOOL ;	//Machine Align Status Against Target Oven for PC (1=Aligned)
    PUSH_PERM : BOOL ;	//Pushing Interlock OK (To Pushers Mc PLC)
    PUSH_LT_MODE : BOOL ;	//Current LT Mode (1-Auto/0-Manual)
    PC_GRP_STATUS : INT ;	//Indicate Whether The Machine Is In The Group Or Out Of Group
    PC_ID : INT ;	//Machine ID for PC
    PC_OVEN_ID_ACT : INT ;	//Oven ID of Present Location for PC
    PUSH_RAM_POS : DINT ;	//Pusher Ram Position
    SPAR_TAG : ARRAY  [0 .. 8 ] OF INT ;
   END_STRUCT ;
   GC_HMI_TAG : STRUCT
    GC_RF_Communicating : BOOL ;	//RF communication OK
    GC_Enc_STATUS : BOOL ;	//Encoder Status for DE
    GC_RF_STATUS : BOOL ;	//RF Modem Status for DE
    GC_AutoSpot_STATUS : BOOL ;	//AutoSPOT  Status for DE
    GC_FLD_STATUS : BOOL ;	//Field Devices (ENC, plc, AutoSPOT, & RF) Status Combined
    GC_MCH_STATUS : BOOL ;	//Machine Health & Operation Status for DE
    GC_ALIGN_STATUS : BOOL ;	//Machine Align Status Against Target Oven for DE (1=Aligned)
    GC_PERM : BOOL ;	//Manual confirmation (Ready for coke)
    GC_SPEED : BOOL ;	//Guide car speed feedback
    GC_LT_MODE : BOOL ;	//Current LT Mode (1-Auto/0-Manual)
    GC_GRP_STATUS : INT ;	//Indicate Whether The Machine Is In The Group Or Out Of Group
    GC_ID : INT ;	//Machine ID for DE
    GC_OVEN_ID_ACT : INT ;	//Oven ID of Present Location for DE
    SPAR_TAG : ARRAY  [0 .. 8 ] OF INT ;
   END_STRUCT ;
   CC_HMI_TAG : STRUCT
    CC_RF_Communicating : BOOL ;	//RF communication OK
    CC_Enc_STATUS : BOOL ;	//Encoder Status for CC
    CC_RF_STATUS : BOOL ;	//RF Modem Status for CC
    CC_AutoSpot_STATUS : BOOL ;	//AutoSPOT  Status for CC
    CC_CHARGING_COMPLETE : BOOL ;	//Field Devices (ENC, plc, AutoSPOT, & RF) Status Combined
    CC_MCH_STATUS : BOOL ;	//Machine Health & Operation Status for CC
    CC_ALIGN_STATUS : BOOL ;	//Machine Align Status Against Target Oven for CC
    CC_PERM : BOOL ;	//Manual confirmation (leveling to  start)
    CC_LT_MODE : BOOL ;	//Current LT Mode (1-Auto/0-Manual)
    LEVLLING_PERM : BOOL ;	//LEVLLEING in progress
    CC_GRP_STATUS : INT ;	//Indicate Whether The Machine Is In The Group Or Out Of Group
    CC_ID : INT ;	//Machine ID for CC
    CC_OVEN_ID_ACT : INT ;	//Oven ID of Present Location for CC
    SPAR_TAG : ARRAY  [0 .. 8 ] OF INT ;
   END_STRUCT ;
   QL_HMI_TAG : STRUCT
    QL_RF_Communicating : BOOL ;	//RF communication OK
    QL_Enc_STATUS : BOOL ;	//Encoder Status for QL
    QL_RF_STATUS : BOOL ;	//RF Modem Status for QL
    QL_AutoSpot_STATUS : BOOL ;	//AutoSPOT  Status for QL
    QL_FLD_STATUS : BOOL ;	//Field Devices (ENC, plc, AutoSPOT, & RF) Status Combined
    QL_MCH_STATUS : BOOL ;	//Machine Health & Operation Status for QL
    QL_ALIGN_STATUS : BOOL ;	// (1=Aligned)
    QL_PERM : BOOL ;	//Manual confirmation (QL is ready to receive coke)
    QL_LT_MODE : BOOL ;	//Current LT Mode (1-Auto/0-Manual)
    QL_COB1 : BOOL ;	//Request for moving battery#1
    QL_COB2 : BOOL ;	//Request for moving battery#2
    QL_GRP_STATUS : INT ;	//Indicate Whether The Machine Is In The Group Or Out Of Group(1-bat#1,2-bat#2,)
    QL_ID : INT ;	//Machine ID for QL
    QL_OVEN_ID_ACT : INT ;	//Oven ID of Present Location for QL
    QL_POS : DINT ;	//Location of QL During Loco Synchronization
    SPAR_TAG : ARRAY  [0 .. 8 ] OF INT ;
   END_STRUCT ;
   L2_HMI_TAG : STRUCT
    L2_TOP_FIVE_SCH_OVEN1 : INT ;	//Pushing Schedule (Oven ID)
    L2_TOP_FIVE_SCH_OVEN2 : INT ;	//------------ " ------------
    L2_TOP_FIVE_SCH_OVEN3 : INT ;	//------------ " ------------
    L2_TOP_FIVE_SCH_OVEN4 : INT ;	//------------ " ------------
    L2_TOP_FIVE_SCH_OVEN5 : INT ;	//------------ " ------------
    L2_SCH_ACTON_MOM1 : STRING  [1 ];	//Action Type
    L2_SCH_ACTON_MOM2 : STRING  [1 ];	//------------ " ------------
    L2_SCH_ACTON_MOM3 : STRING  [1 ];	//------------ " ------------
    L2_SCH_ACTON_MOM4 : STRING  [1 ];	//------------ " ------------
    L2_SCH_ACTON_MOM5 : STRING  [1 ];	//------------ " ------------
    L2_SCH_OVEN_ACTION_TIME1 : STRING  [17 ];	//Action Time
    L2_SCH_OVEN_ACTION_TIME2 : STRING  [17 ];	//------------ " ------------
    L2_SCH_OVEN_ACTION_TIME3 : STRING  [17 ];	//------------ " ------------
    L2_SCH_OVEN_ACTION_TIME4 : STRING  [17 ];	//------------ " ------------
    L2_SCH_OVEN_ACTION_TIME5 : STRING  [17 ];	//------------ " ------------
    PUSHED_OVN : INT ;	//For Updating L-II
    PUSHED_AT : INT ;	//For Updating L-II
    LEVELLED_OVN : INT ;	//For Updating L-II
    LEVELLED_AT : INT ;	//For Updating L-II
    ACK_MODE_SEL : BOOL ;	//PLC Confirms The Change Over From Auto To Manual & Vis Versa
    MCH_DIS_DIFF : DINT ;	//Distance Reaming (In MM) For Target Oven
    PC_OVEN_ID_TAR : INT ;	//Oven ID of Target Location for PC
    PC_OVEN_ID_LAST : INT ;	//Oven ID of Last Operation
    PC_OPERATION_LAST : STRING  [1 ];	//Last Operation (PUSH, LEVEL, …)
    PC_DATETIME_LAST : STRING  [17 ];	//Actual Pushing/Levelling Time for Last Operation
    PC_OVEN_ID_NEXT : INT ;	//Oven ID of Next Operation
    PC_OPERATION_NEXT : STRING  [1 ];	//Next Operation (PUSH, LEVEL, …)
    PC_DATETIME_NEXT : STRING  [17 ];	//Planned Pushing/Levelling Time for Next Operation
    PC_NEXT_OPR_INPROGRESS : BOOL ;	//NEXT OPERATION IN PROGRESS (LAST COMPLETED)
    PC_LAST_PUSHED_OVEN : INT ;	//PC_LAST_PUSHED_OVEN
    CC_LAST_CHARGED_OVEN : INT ;	//CC_LAST_CHARGED_OVEN
    PC_PUSH_START : BOOL ;	//PC_PUSH_START
    SPAR_TAG : ARRAY  [0 .. 8 ] OF DINT ;
    stat : BYTE ;
   END_STRUCT ;
  END_STRUCT ;	
BEGIN
END_DATA_BLOCK

DATA_BLOCK "DB:User"	// DB 36
VERSION : 0.1
  STRUCT
   PC_1_Status_Store : BOOL ;
   PC_2_Status_Store : BOOL ;
   PC_1_2_Status_Compare : BOOL ;
   CC_1_Status_Store : BOOL ;
   CC_2_Status_Store : BOOL ;
   CC_1_2_Status_Compare : BOOL ;
   GC_1_Status_Store : BOOL ;
   GC_2_Status_Store : BOOL ;
   GC_1_2_Status_Compare : BOOL ;
   QL_1_Status_Store : BOOL ;
   QL_2_Status_Store : BOOL ;
   QL_1_2_Status_Compare : BOOL ;
   Pulse_1 : BOOL ;
   Pulse_2 : BOOL ;
   Pulse_3 : BOOL ;
   Pulse_4 : BOOL ;
   PC_Communication_1 : BOOL ;
   PC_Communication_0 : BOOL ;
   PC_Communication_ERR : BOOL ;
   CC_Communication_1 : BOOL ;
   CC_Communication_0 : BOOL ;
   CC_Communication_ERR : BOOL ;
   GC_Communication_1 : BOOL ;
   GC_Communication_0 : BOOL ;
   GC_Communication_ERR : BOOL ;
   QL_Communication_1 : BOOL ;
   QL_Communication_0 : BOOL ;
   QL_Communication_ERR : BOOL ;
   Pulse_5 : BOOL ;
   Pulse_6 : BOOL ;
   PC_RxDT_Trigger : BOOL ;
   CC_RxDT_Trigger : BOOL ;
   GC_RxDT_Trigger : BOOL ;
   QL_RxDT_Trigger : BOOL ;
   F1_COB_2 : BOOL ;
   Offline_COB_1 : BOOL ;
   Modem_FrQ_Don : BOOL ;
   Modem_FrQ_Err : BOOL ;
   Pulse_7 : BOOL ;
   PC_OvenID_Compar : BOOL ;
   CC_OvenID_Compar : BOOL ;
   GC_OvenID_Compar : BOOL ;
   QL_OvenID_Compar : BOOL ;
   Pulse_8 : BOOL ;
   Pulse_9 : BOOL ;
   PC_POS_OK_1 : BOOL ;
   GC_POS_OK_1 : BOOL ;
   QL_POS_OK_1 : BOOL ;
   PUSHING_COMPLITE_OK : BOOL ;
   Curr_Trg : BOOL ;
   PC_MC_ID_Status : INT ;
   CC_MC_ID_Status : INT ;
   GC_MC_ID_Status : INT ;
   QL_MC_ID_Status : INT ;
   PC_REL_VAL : INT ;
   CC_REL_VAL : INT ;
   GC_REL_VAL : INT ;
   QL_REL_VAL : INT ;
   L2_REL_VAL : INT ;
   PC_STat_REL_VAL : INT ;
   CC_STat_REL_VAL : INT ;
   GC_STat_REL_VAL : INT ;
   QL_STat_REL_VAL : INT ;
   CC_TAR_OVEN_1 : INT ;
   PC_TAR_OVEN_1 : INT ;
   CC_TAR_OVEN_2 : INT ;
   PC_TAR_OVEN_2 : INT ;
   CC_TAR_OVEN_3 : INT ;
   PC_TAR_OVEN_3 : INT ;
   CC_TAR_OVEN_4 : INT ;
   PC_TAR_OVEN_4 : INT ;
   CC_TAR_OVEN_5 : INT ;
   PC_TAR_OVEN_5 : INT ;
   CR_REL_VAL : INT ;
   Push_Curr_REL_VAL : INT ;
   STAT_INT0112 : INT ;
   STAT_INT023 : INT ;
   STAT_INT0113 : INT ;
   STAT_INT024 : INT ;
   STAT_INT0114 : INT ;
   STAT_INT025 : INT ;
   STAT_INT0115 : INT ;
   STAT_INT026 : INT ;
   STAT_INT0116 : INT ;
   STAT_INT027 : INT ;
   STAT_INT0117 : INT ;
   STAT_WORD0 : WORD ;
   STAT_WORD1 : WORD ;
   STAT_WORD2 : WORD ;
   STAT_WORD3 : WORD ;
   STAT_WORD03 : WORD ;
   STAT_WORD012 : WORD ;
   STAT_WORD04 : WORD ;
   STAT_WORD013 : WORD ;
   STAT_WORD05 : WORD ;
   STAT_WORD014 : WORD ;
   STAT_WORD06 : WORD ;
   STAT_WORD015 : WORD ;
   STAT_WORD07 : WORD ;
   STAT_WORD016 : WORD ;
   STAT_WORD08 : WORD ;
   STAT_WORD017 : WORD ;
   STAT_WORD09 : WORD ;
   STAT_WORD018 : WORD ;
   STAT_WORD010 : WORD ;
   STAT_WORD019 : WORD ;
   PULSE_50 : BOOL ;
   PULSE_51 : BOOL ;
   PULSE_52 : BOOL ;
   PULSE_53 : BOOL ;
   PULSE_54 : BOOL ;
   PULSE_55 : BOOL ;
   PULSE_56 : BOOL ;
   PULSE_57 : BOOL ;
   PULSE_58 : BOOL ;
   PULSE_59 : BOOL ;
   PULSE_60 : BOOL ;
   PULSE_61 : BOOL ;
   PULSE_62 : BOOL ;
   PULSE_63 : BOOL ;
   PULSE_64 : BOOL ;
   PULSE_65 : BOOL ;
   PULSE_66 : BOOL ;
   PULSE_67 : BOOL ;
   PULSE_68 : BOOL ;
   PULSE_70 : BOOL ;
   PULSE_71 : BOOL ;
   PULSE_72 : BOOL ;
   PULSE_73 : BOOL ;
   PULSE_74 : BOOL ;
   PULSE_75 : BOOL ;
   PULSE_76 : BOOL ;
   PULSE_77 : BOOL ;
   PULSE_78 : BOOL ;
   PULSE_79 : BOOL ;
   PULSE_80 : BOOL ;
   PULSE_81 : BOOL ;
   PULSE_82 : BOOL ;
   PULSE_83 : BOOL ;
   PULSE_84 : BOOL ;
   PULSE_85 : BOOL ;
   PULSE_86 : BOOL ;
   PULSE_87 : BOOL ;
   PULSE_88 : BOOL ;
   PULSE_89 : BOOL ;
   PULSE_90 : BOOL ;
   PC_POS_OK_2 : BOOL ;
   GC_POS_OK_2 : BOOL ;
   QL_POS_OK_2 : BOOL ;
   PC_POS_OK_3 : BOOL ;
   GC_POS_OK_3 : BOOL ;
   QL_POS_OK_3 : BOOL ;
   PC_POS_OK_4 : BOOL ;
   GC_POS_OK_4 : BOOL ;
   QL_POS_OK_4 : BOOL ;
   PC_POS_OK_5 : BOOL ;
   GC_POS_OK_5 : BOOL ;
   QL_POS_OK_5 : BOOL ;
   PULSE_5052 : BOOL ;
   PULSE_5053 : BOOL ;
   PULSE_5054 : BOOL ;
   PULSE_5055 : BOOL ;
   PULSE_5056 : BOOL ;
   PULSE_5057 : BOOL ;
   PULSE_5058 : BOOL ;
   PULSE_5059 : BOOL ;
   PULSE_5060 : BOOL ;
   STAT_WORD0110 : WORD ;
   STAT_WORD021 : WORD ;
   STAT_WORD0111 : WORD ;
   STAT_WORD022 : WORD ;
   STAT_WORD0112 : WORD ;
   STAT_WORD023 : WORD ;
   STAT_WORD0113 : WORD ;
   STAT_WORD024 : WORD ;
   STAT_WORD0114 : WORD ;
   STAT_WORD025 : WORD ;
   SHOW_P_1 : BOOL ;	//SHOW_P_1_for_sch
   SHOW_C_1 : BOOL ;	//SHOW_C_1_for_sch
   SHOW_P_2 : BOOL ;	//SHOW_P_2_for_sch
   SHOW_C_2 : BOOL ;	//SHOW_C_2_for_sch
   post_plse_use : BOOL ;	//post_plse_use
   push_count : INT ;	//push_count
   sch_a : INT ;
   COB_2_FREQ : BOOL ;	//BATT#2 FREQ SELECTION BIT
  END_STRUCT ;	
BEGIN
END_DATA_BLOCK

DATA_BLOCK "DB:InitializationRxBuffe"	// DB 39
VERSION : 0.1
  STRUCT
   RCVBufferInitialization : ARRAY  [1 .. 500 ] OF //Recived Buffer Reset
   BYTE ;
  END_STRUCT ;	
BEGIN
END_DATA_BLOCK

DATA_BLOCK "DB:SndWork DB RS232C"	// DB 40
//P_SND_RK Work-DB 
//
VERSION : 0.1
  STRUCT
   P_SND_ASCII_REQ : BOOL ;
   P_SND_ASCII_R : BOOL ;
   P_SND_ASCII_CommoN_REQ : BOOL ;
   STATE1 : BOOL ;
   P_SND_ASCII_DONE : BOOL ;
   P_SND_ASCII_ERROR : BOOL ;
   STATE2 : BOOL ;
   STATE3 : BOOL ;
   P_SND_ASCII_WORK_LADD : INT ;
   P_SND_ASCII_WORK_DB_N : INT ;
   P_SND_ASCII_WORK_DBB_NO : INT ;
   P_SND_ASCII_WORK_LEN : INT ;
   STATE4 : WORD ;
   P_SND_ASCII_WORK_STATUS : WORD ;
   P_SND_WORK_STATUS_SAV : WORD ;
   P_SND_ASCII_COUNTER_OK : WORD ;
   P_SND_ASCII_COUNTER_ERR : WORD ;
   P_SND_ASCII_WORK_DB : ARRAY  [1 .. 80 ] OF BYTE ;
  END_STRUCT ;	
BEGIN
END_DATA_BLOCK

DATA_BLOCK "DB:RevWork DB RS232C"	// DB 41
//P_RCV_RK Work-DB
//
VERSION : 0.1
  STRUCT
   P_RCV_ASCII_EN_R : BOOL ;
   STAT0 : BOOL ;
   STAT1 : BOOL ;
   STAT2 : BOOL ;
   P_RCV_ASCII_NDR : BOOL ;
   P_RCV_ASCII_ERROR : BOOL ;
   STAT3 : BOOL ;
   STAT4 : BOOL ;
   P_RCV_ASCII_WORK_LADDR : INT ;
   P_RCV_ASCII_WORK_DB_NO : INT ;
   P_RCV_ASCII_WORK_DBB_NO : INT ;
   P_RCV_ASCII_WORK_LEN : INT ;
   P_RCV_ASCII_WORK_SAVE_LE : WORD ;
   P_RCV_ASCII_WORK_STATUS : WORD ;
   P_RCV_WORK_STATUS_SAV : WORD ;
   STAT5 : WORD ;
   P_RCV_ASCII_WORK_CNT_OK : WORD ;
   P_RCV_ASCII_WORK_CNT_ERR : WORD ;
   P_RCV_ASCII_WORK_DB : ARRAY  [1 .. 80 ] OF BYTE ;
  END_STRUCT ;	
BEGIN
END_DATA_BLOCK

DATA_BLOCK "testng_4_ram_curent_fc45"	// DB 45
VERSION : 0.1
  STRUCT
   DB_VAR : INT ;	//Temporary placeholder variable
  END_STRUCT ;	
BEGIN
END_DATA_BLOCK

DATA_BLOCK "FOR_FC-45-OFFLINE"	// DB 46
VERSION : 0.1
  STRUCT
   START : BOOL ;	//Temporary placeholder variable
   STOP : BOOL ;
   HALF_SEC_TIMER : BOOL ;
   COUNT_RESET : BOOL ;
   COUNT_VALUE : WORD ;
   DISP_COB : BOOL ;
   DISP_OVEN : BOOL ;
   DISP_BATT : BOOL ;
   DISP_3 : BOOL ;
   DISP_1 : BOOL ;
   DISP_ONCE_TIME : BOOL ;
   DISP_M : BOOL ;
   DISP_B : BOOL ;
   DISP : BOOL ;
   DISP_T1 : BOOL ;
   DISP_A1 : BOOL ;
   DISP_T2 : BOOL ;
   DISP_A2 : BOOL ;
   offline_cc_id : INT ;	//offline_cc_id
   OFF_LAST_CHRG_OVEN : INT ;	//OFF_LAST_CHRG_OVEN
   POST_PULSE : BOOL ;	//POST_PULSE
   CHRG_1_OFFLINE : BOOL ;	//CHRG_1_OFFLINE
   CHRG_2_OFFLINE : BOOL ;	//CHRG_2_OFFLINE
   CHRG_3_OFFLINE : BOOL ;	//CHRG_3_OFFLINE
  END_STRUCT ;	
BEGIN
END_DATA_BLOCK

DATA_BLOCK "IDB_RS232_RM_ChgFreq_SND"	// DB 50
AUTHOR : SIMATIC
FAMILY : CP341
VERSION : 0.0
"P_SND_ASCII"
BEGIN
END_DATA_BLOCK

DATA_BLOCK "IDB_RS232_RM_ChgFreq_RCV"	// DB 51
AUTHOR : SIMATIC
FAMILY : CP341
VERSION : 0.0
"P_RCV_ASCII"
BEGIN
END_DATA_BLOCK

DATA_BLOCK "IDB_RS485_AutoSPOT_RCV"	// DB 80
AUTHOR : SIMATIC
FAMILY : CP341
VERSION : 0.0
"P_RCV_ASCII"
BEGIN
END_DATA_BLOCK

DATA_BLOCK "DB:USE"	// DB 100
VERSION : 0.1
  STRUCT
   DP_SEND_DONE : BOOL ;
   DP_SEND_ERROR : BOOL ;
   DP_RECEIVE_NDR : BOOL ;
   DP_RECEIVE_ERROR : BOOL ;
   FC31_ENABLE : BOOL ;
   PULSE_1 : BOOL ;
   Change_Frequency : BOOL ;
   PULSE_2 : BOOL ;
   PULSE_3 : BOOL ;
   Initializing : BOOL ;
   PULSE_4 : BOOL ;
   Chang_Frq_Respons_OK : BOOL ;
   Chang_Frq_Respons_ERR : BOOL ;
   Chang_Frq_Respons_SUCC : BOOL ;
   Chang_Frq_Req_ERR : BOOL ;
   Save_Frq_Respons_OK : BOOL ;
   Save_Frq_Respons_ERR : BOOL ;
   Freq_Chang_Req_Succ : BOOL ;
   Freq_Chang_Req_Err : BOOL ;
   Freq_Setting_Inform : BOOL ;
   Offline_Freq_Chang : BOOL ;
   PULSE_5 : BOOL ;
   PULSE_6 : BOOL ;
   PULSE_7 : BOOL ;
   FRequency_Trigger : BOOL ;
   Event_Trigger : BOOL ;
   PULSE_8 : BOOL ;
   PULSE_9 : BOOL ;
   PULSE_10 : BOOL ;
   Comprator5 : BOOL ;
   PULSE_11 : BOOL ;
   PULSE_12 : BOOL ;
   CP_Communication_Err : BOOL ;
   PULSE_13 : BOOL ;
   PULSE_14 : BOOL ;
   PULSE_15 : BOOL ;
   PULSE_16 : BOOL ;
   PULSE_17 : BOOL ;
   PULSE_18 : BOOL ;
   StatBit39 : BOOL ;
   DP_RECEIVE_DPSTATUS : BYTE ;
   StatByte1 : BYTE ;
   StatByte2 : BYTE ;
   StatByte3 : BYTE ;
   StatByte4 : BYTE ;
   StatByte5 : BYTE ;
   StatByte6 : BYTE ;
   StatByte7 : BYTE ;
   StatByte8 : BYTE ;
   StatByte9 : BYTE ;
   StatByte10 : BYTE ;
   StatByte11 : BYTE ;
   StatByte12 : BYTE ;
   StatByte13 : BYTE ;
   StatByte14 : BYTE ;
   StatByte15 : BYTE ;
   StatByte16 : BYTE ;
   StatByte17 : BYTE ;
   StatByte18 : BYTE ;
   StatByte19 : BYTE ;
   StatByte20 : BYTE ;
   DP_SEND_STATUS : WORD ;
   DP_RECEIVE_STATUS : WORD ;
   StatWord2 : WORD ;
   StatWord3 : WORD ;
   StatWord4 : WORD ;
   StatWord5 : WORD ;
   StatWord6 : WORD ;
   StatWord7 : WORD ;
   StatWord8 : WORD ;
   StatWord9 : WORD ;
   StatWord10 : WORD ;
   StatWord11 : WORD ;
   StatWord12 : WORD ;
   StatWord13 : WORD ;
   StatWord14 : WORD ;
   StatWord15 : WORD ;
   StatWord16 : WORD ;
   StatWord17 : WORD ;
   StatWord18 : WORD ;
   StatWord19 : WORD ;
   StatWord20 : WORD ;
   StatDWord0 : DWORD ;
   StatDWord1 : DWORD ;
   StatDWord2 : DWORD ;
   StatDWord3 : DWORD ;
   StatDWord4 : DWORD ;
   StatDWord5 : DWORD ;
   StatDWord6 : DWORD ;
   StatDWord7 : DWORD ;
   StatDWord8 : DWORD ;
   StatDWord9 : DWORD ;
   StatDWord10 : DWORD ;
   SELECT_BATT : INT  := 1;
   Schedule_Adder : INT ;
   Initialise_SFC20_1 : INT ;
   Initialise_SFC20_2 : INT ;
   StatInt4 : INT ;
   StatInt5 : INT ;
   StatInt6 : INT ;
   StatInt7 : INT ;
   StatInt8 : INT ;
   StatInt9 : INT ;
   StatInt10 : INT ;
   StatDInt0 : DINT ;
   StatDInt1 : DINT ;
   StatDInt2 : DINT ;
   StatDInt3 : DINT ;
   StatDInt4 : DINT ;
   StatDInt5 : DINT ;
   StatDInt6 : DINT ;
   StatDInt7 : DINT ;
   StatDInt8 : DINT ;
   StatDInt9 : DINT ;
   StatDInt10 : DINT ;
   Encode_Calc1 : REAL ;
   Encode_Calc2 : REAL ;
   StatReal2 : REAL ;
   StatReal3 : REAL ;
   StatReal4 : REAL ;
   StatReal5 : REAL ;
   StatReal6 : REAL ;
   StatReal7 : REAL ;
   StatReal8 : REAL ;
   StatReal9 : REAL ;
   StatReal10 : REAL ;
  END_STRUCT ;	
BEGIN
   SELECT_BATT := 1;
END_DATA_BLOCK

ORGANIZATION_BLOCK "CYCL_EXC"	// OB 1
TITLE = "Main Program Sweep (Cycle)"
VERSION : 0.1
VAR_TEMP
  OB1_EV_CLASS : BYTE ;	//Bits 0-3 = 1 (Coming event), Bits 4-7 = 1 (Event class 1)
  OB1_SCAN_1 : BYTE ;	//1 (Cold restart scan 1 of OB 1), 3 (Scan 2-n of OB 1)
  OB1_PRIORITY : BYTE ;	//Priority of OB Execution
  OB1_OB_NUMBR : BYTE ;	//1 (Organization block 1, OB1)
  OB1_RESERVED_1 : BYTE ;	//Reserved for system
  OB1_RESERVED_2 : BYTE ;	//Reserved for system
  OB1_PREV_CYCLE : INT ;	//Cycle time of previous OB1 scan (milliseconds)
  OB1_MIN_CYCLE : INT ;	//Minimum cycle time of OB1 (milliseconds)
  OB1_MAX_CYCLE : INT ;	//Maximum cycle time of OB1 (milliseconds)
  OB1_DATE_TIME : DATE_AND_TIME ;	//Date and time OB1 started
END_VAR
BEGIN
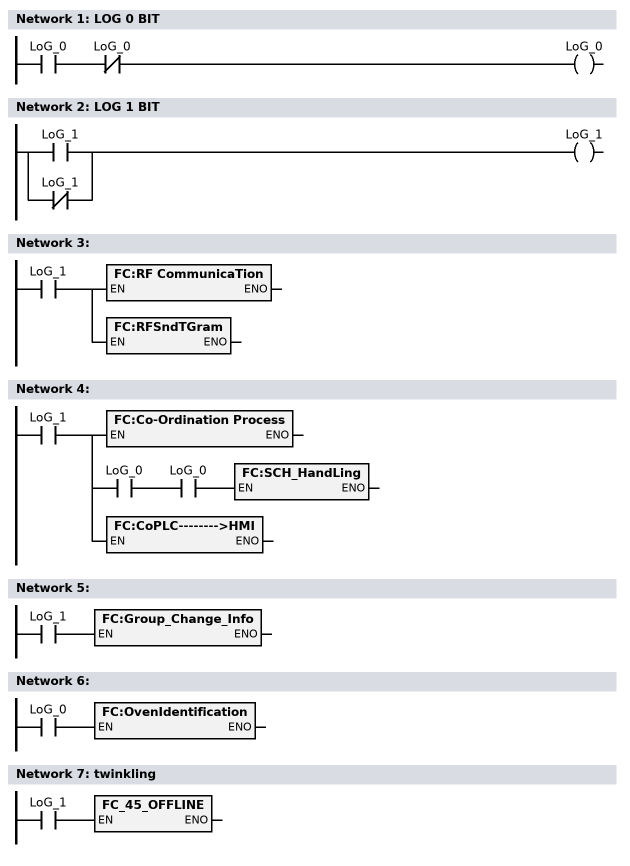
NETWORK
TITLE = LOG 0 BIT
      A     "LoG_0";
      AN    "LoG_0";
      =     "LoG_0";
NETWORK
TITLE = LOG 1 BIT
      O     "LoG_1";
      ON    "LoG_1";
      =     "LoG_1";
NETWORK
TITLE =
      A     "LoG_1";
      =     L 20.0;
      A     L 20.0;
      JNB   _001;
      CALL  "FC:RF CommunicaTion";
_001: NOP   0;
      A     L 20.0;
      JNB   _002;
      CALL  "FC:RFSndTGram";
_002: NOP   0;
NETWORK
TITLE =
      A     "LoG_1";
      =     L 20.0;
      A     L 20.0;
      JNB   _003;
      CALL  "FC:Co-Ordination Process";
_003: NOP   0;
      A     L 20.0;
      A     "LoG_0";
      A     "LoG_0";
      JNB   _004;
      CALL  "FC:SCH_HandLing";
_004: NOP   0;
      A     L 20.0;
      JNB   _005;
      CALL  "FC:CoPLC-------->HMI";
_005: NOP   0;
NETWORK
TITLE =
      A     "LoG_1";
      JNB   _006;
      CALL  "FC:Group_Change_Info";
_006: NOP   0;
NETWORK
TITLE =
      A     "LoG_0";
      JNB   _007;
      CALL  "FC:OvenIdentification";
_007: NOP   0;
NETWORK
TITLE = twinkling
      A     "LoG_1";
      JNB   _008;
      CALL  "FC_45_OFFLINE";
_008: NOP   0;
END_ORGANIZATION_BLOCK

ORGANIZATION_BLOCK "PROG_ERR"	// OB 121
TITLE = "Programming Error"
VERSION : 0.1
VAR_TEMP
  OB121_EV_CLASS : BYTE ;	//16#25, Event class 2, Entering event state, Internal fault event
  OB121_SW_FLT : BYTE ;	//16#XX Software programming fault
  OB121_PRIORITY : BYTE ;	//Priority of OB Execution
  OB121_OB_NUMBR : BYTE ;	//121 (Organization block 121, OB121)
  OB121_BLK_TYPE : BYTE ;	//16#88/8A/8B/8C/8E Type of block fault occured in
  OB121_RESERVED_1 : BYTE ;	//Reserved for system
  OB121_FLT_REG : WORD ;	//16#XX Specific register that caused fault
  OB121_BLK_NUM : WORD ;	//Number of block that programming fault occured in
  OB121_PRG_ADDR : WORD ;	//Address in block where programming fault occured
  OB121_DATE_TIME : DATE_AND_TIME ;	//Date and time OB121 started
END_VAR
BEGIN
NETWORK
TITLE =
END_ORGANIZATION_BLOCK

ORGANIZATION_BLOCK "MOD_ERR"	// OB 122
TITLE = "Module Access Error"
VERSION : 0.1
VAR_TEMP
  OB122_EV_CLASS : BYTE ;	//16#29, Event class 2, Entering event state, Internal fault event
  OB122_SW_FLT : BYTE ;	//16#XX Software error code
  OB122_PRIORITY : BYTE ;	//Priority of OB Execution
  OB122_OB_NUMBR : BYTE ;	//122 (Organization block 122, OB122)
  OB122_BLK_TYPE : BYTE ;	//16#88/8C/8E Type of block fault occured in
  OB122_MEM_AREA : BYTE ;	//Memory area where access error occured
  OB122_MEM_ADDR : WORD ;	//Memory address where access error occured
  OB122_BLK_NUM : WORD ;	//Block number in which error occured
  OB122_PRG_ADDR : WORD ;	//Program address where error occured
  OB122_DATE_TIME : DATE_AND_TIME ;	//Date and time OB1 started
END_VAR
BEGIN
// (block stored without names or comments; labels and parameter names are numbered)
END_ORGANIZATION_BLOCK
